C01814=1073.007,225.307,-82.417,174.106,27.682,154.920
C01815=1073.013,225.555,-82.444,174.109,27.687,154.920
C01816=1073.019,225.804,-82.469,174.111,27.690,154.921
C01817=1073.025,226.052,-82.496,174.113,27.694,154.921
C01818=1073.031,226.301,-82.522,174.116,27.698,154.922
C01819=1073.036,226.549,-82.549,174.118,27.702,154.923
C01820=1073.043,226.798,-82.574,174.120,27.706,154.923
C01821=1073.048,227.046,-82.601,174.123,27.710,154.924
C01822=1073.054,227.295,-82.627,174.125,27.713,154.924
C01823=1073.060,227.544,-82.652,174.127,27.717,154.925
C01824=1073.066,227.792,-82.679,174.129,27.721,154.926
C01825=1073.072,228.041,-82.705,174.131,27.725,154.926
C01826=1073.078,228.289,-82.731,174.133,27.729,154.927
C01827=1073.084,228.538,-82.757,174.136,27.733,154.927
C01828=1073.089,228.787,-82.783,174.138,27.736,154.928
C01829=1073.096,229.036,-82.810,174.140,27.740,154.929
C01830=1073.102,229.285,-82.835,174.143,27.744,154.929
C01831=1073.107,229.533,-82.862,174.145,27.748,154.930
C01832=1073.113,229.782,-82.888,174.147,27.752,154.930
C01833=1073.119,230.030,-82.914,174.150,27.755,154.931
C01834=1073.125,230.278,-82.941,174.152,27.760,154.932
C01835=1073.131,230.527,-82.967,174.154,27.764,154.932
C01836=1073.136,230.776,-82.993,174.156,27.768,154.933
C01837=1073.142,231.024,-83.020,174.158,27.771,154.933
C01838=1073.148,231.273,-83.046,174.160,27.775,154.934
C01839=1073.153,231.521,-83.073,174.163,27.779,154.935
C01840=1073.159,231.770,-83.099,174.165,27.782,154.935
C01841=1073.165,232.018,-83.126,174.167,27.787,154.936
C01842=1073.170,232.267,-83.152,174.169,27.791,154.936
C01843=1073.177,232.515,-83.178,174.172,27.795,154.937
C01844=1073.183,232.764,-83.205,174.174,27.798,154.938
C01845=1073.189,233.013,-83.231,174.176,27.802,154.938
C01846=1073.195,233.262,-83.257,174.179,27.806,154.939
C01847=1073.200,233.510,-83.284,174.181,27.810,154.939
C01848=1073.206,233.758,-83.311,174.183,27.814,154.940
C01849=1073.212,234.007,-83.337,174.186,27.818,154.941
C01850=1073.218,234.255,-83.364,174.188,27.821,154.941
C01851=1073.223,234.504,-83.390,174.190,27.825,154.942
C01852=1073.229,234.752,-83.417,174.193,27.829,154.943
C01853=1073.235,235.001,-83.443,174.195,27.833,154.943
C01854=1073.244,235.416,-83.489,174.198,27.839,154.944
C01855=1073.254,235.831,-83.533,174.202,27.846,154.945
C01856=1073.264,236.245,-83.577,174.206,27.852,154.946
C01857=1073.273,236.660,-83.623,174.210,27.859,154.947
C01858=1073.279,236.908,-83.649,174.212,27.863,154.948
C01859=1073.285,237.157,-83.676,174.214,27.867,154.948
C01860=1073.291,237.405,-83.703,174.217,27.871,154.949
C01861=1073.296,237.653,-83.729,174.219,27.874,154.950
C01862=1073.303,237.902,-83.756,174.221,27.878,154.950
C01863=1073.309,238.151,-83.783,174.224,27.882,154.951
C01864=1073.314,238.399,-83.809,174.226,27.886,154.951
C01865=1073.320,238.648,-83.836,174.228,27.890,154.952
C01866=1073.327,238.897,-83.863,174.231,27.894,154.953
C01867=1073.332,239.145,-83.890,174.233,27.897,154.953
C01868=1073.337,239.394,-83.917,174.235,27.901,154.954
C01869=1073.343,239.642,-83.944,174.238,27.905,154.954
C01870=1073.350,239.891,-83.971,174.240,27.909,154.955
C01871=1073.355,240.139,-83.997,174.242,27.913,154.956
C01872=1073.361,240.387,-84.025,174.245,27.917,154.956
C01873=1073.367,240.636,-84.051,174.247,27.920,154.957
C01874=1073.373,240.885,-84.079,174.249,27.924,154.957
C01875=1073.379,241.133,-84.106,174.252,27.928,154.958
C01876=1073.384,241.382,-84.132,174.254,27.932,154.959
C01877=1073.390,241.629,-84.160,174.257,27.936,154.959
C01878=1073.397,241.878,-84.187,174.259,27.940,154.960
C01879=1073.402,242.127,-84.214,174.261,27.943,154.960
C01880=1073.408,242.375,-84.241,174.264,27.947,154.961
C01881=1073.414,242.624,-84.268,174.266,27.951,154.962
C01882=1073.420,242.872,-84.295,174.268,27.955,154.962
C01883=1073.425,243.121,-84.322,174.271,27.959,154.963
C01884=1073.431,243.369,-84.350,174.273,27.963,154.963
C01885=1073.438,243.618,-84.377,174.275,27.967,154.964
C01886=1073.443,243.866,-84.404,174.278,27.971,154.965
C01887=1073.449,244.114,-84.431,174.280,27.975,154.965
C01888=1073.454,244.364,-84.459,174.282,27.978,154.966
C01889=1073.460,244.612,-84.485,174.285,27.982,154.966
C01890=1073.466,244.860,-84.513,174.287,27.986,154.967
C01891=1073.472,245.109,-84.540,174.289,27.990,154.968
C01892=1073.478,245.357,-84.568,174.292,27.994,154.968
C01893=1073.483,245.605,-84.595,174.294,27.998,154.969
C01894=1073.490,245.854,-84.623,174.296,28.002,154.970
C01895=1073.495,246.103,-84.650,174.300,28.005,154.970
C01896=1073.500,246.351,-84.677,174.302,28.009,154.971
C01897=1073.507,246.599,-84.704,174.304,28.013,154.971
C01898=1073.512,246.848,-84.732,174.307,28.017,154.972
C01899=1073.518,247.096,-84.759,174.309,28.021,154.972
C01900=1073.524,247.344,-84.787,174.312,28.025,154.973
C01901=1073.529,247.593,-84.815,174.314,28.029,154.974
C01902=1073.535,247.841,-84.842,174.316,28.033,154.974
C01903=1073.541,248.090,-84.869,174.319,28.036,154.975
C01904=1073.547,248.338,-84.897,174.321,28.040,154.976
C01905=1073.552,248.587,-84.924,174.323,28.045,154.976
C01906=1073.562,248.995,-84.970,174.327,28.051,154.977
C01907=1073.571,249.403,-85.015,174.331,28.057,154.978
C01908=1073.581,249.812,-85.061,174.335,28.064,154.979
C01909=1073.590,250.219,-85.107,174.339,28.070,154.980
C01910=1073.595,250.468,-85.134,174.341,28.074,154.981
C01911=1073.601,250.716,-85.161,174.344,28.078,154.982
C01912=1073.607,250.965,-85.190,174.346,28.082,154.982
C01913=1073.613,251.213,-85.218,174.348,28.086,154.983
C01914=1073.619,251.462,-85.245,174.351,28.090,154.983
C01915=1073.624,251.710,-85.273,174.353,28.094,154.984
C01916=1073.630,251.958,-85.301,174.356,28.097,154.985
C01917=1073.636,252.206,-85.328,174.359,28.101,154.985
C01918=1073.641,252.455,-85.356,174.361,28.105,154.986
C01919=1073.647,252.704,-85.384,174.363,28.109,154.986
C01920=1073.653,252.951,-85.411,174.366,28.113,154.987
C01921=1073.659,253.200,-85.440,174.368,28.117,154.988
C01922=1073.665,253.448,-85.468,174.371,28.121,154.988
C01923=1073.671,253.697,-85.495,174.373,28.125,154.989
C01924=1073.677,253.945,-85.523,174.375,28.128,154.989
C01925=1073.683,254.193,-85.552,174.378,28.132,154.990
C01926=1073.688,254.442,-85.579,174.380,28.136,154.991
C01927=1073.694,254.691,-85.607,174.383,28.140,154.991
C01928=1073.700,254.939,-85.635,174.386,28.144,154.992
C01929=1073.706,255.187,-85.663,174.388,28.148,154.993
C01930=1073.712,255.436,-85.691,174.390,28.152,154.993
C01931=1073.718,255.684,-85.719,174.393,28.156,154.994
C01932=1073.724,255.933,-85.747,174.395,28.160,154.994
C01933=1073.729,256.181,-85.775,174.398,28.164,154.995
C01934=1073.735,256.429,-85.803,174.400,28.167,154.996
C01935=1073.741,256.677,-85.831,174.402,28.171,154.996
C01936=1073.747,256.926,-85.859,174.406,28.175,154.997
C01937=1073.753,257.175,-85.887,174.408,28.179,154.997
C01938=1073.758,257.423,-85.915,174.410,28.183,154.998
C01939=1073.765,257.671,-85.944,174.413,28.187,154.999
C01940=1073.771,257.919,-85.972,174.415,28.190,154.999
C01941=1073.776,258.167,-86.000,174.418,28.194,155.000
C01942=1073.782,258.416,-86.028,174.420,28.198,155.000
C01943=1073.788,258.664,-86.056,174.422,28.202,155.001
C01944=1073.794,258.913,-86.084,174.426,28.206,155.002
C01945=1073.800,259.161,-86.112,174.428,28.210,155.002
C01946=1073.806,259.409,-86.141,174.430,28.214,155.003
C01947=1073.812,259.657,-86.169,174.433,28.217,155.003
C01948=1073.818,259.906,-86.198,174.435,28.221,155.004
C01949=1073.824,260.154,-86.225,174.438,28.225,155.005
C01950=1073.830,260.403,-86.253,174.440,28.229,155.005
C01951=1073.836,260.651,-86.282,174.443,28.233,155.006
C01952=1073.842,260.899,-86.310,174.446,28.237,155.006
C01953=1073.847,261.148,-86.339,174.448,28.241,155.007
C01954=1073.854,261.396,-86.368,174.450,28.245,155.008
C01955=1073.860,261.644,-86.395,174.453,28.248,155.008
C01956=1073.866,261.892,-86.423,174.455,28.252,155.009
C01957=1073.872,262.140,-86.452,174.459,28.256,155.009
C01958=1073.881,262.547,-86.499,174.463,28.262,155.010
C01959=1073.891,262.952,-86.545,174.467,28.268,155.011
C01960=1073.902,263.357,-86.591,174.471,28.275,155.012
C01961=1073.911,263.764,-86.638,174.475,28.281,155.013
C01962=1073.917,264.011,-86.666,174.477,28.285,155.014
C01963=1073.923,264.260,-86.695,174.480,28.289,155.015
C01964=1073.929,264.508,-86.724,174.483,28.293,155.015
C01965=1073.934,264.756,-86.752,174.485,28.297,155.016
C01966=1073.941,265.004,-86.781,174.488,28.300,155.016
C01967=1073.946,265.253,-86.810,174.490,28.304,155.017
C01968=1073.952,265.502,-86.839,174.493,28.309,155.018
C01969=1073.957,265.750,-86.867,174.496,28.312,155.018
C01970=1073.964,265.998,-86.896,174.498,28.316,155.019
C01971=1073.970,266.246,-86.925,174.500,28.320,155.019
C01972=1073.976,266.495,-86.953,174.503,28.324,155.020
C01973=1073.981,266.742,-86.982,174.505,28.328,155.021
C01974=1073.987,266.991,-87.011,174.508,28.332,155.021
C01975=1073.993,267.239,-87.040,174.511,28.336,155.022
C01976=1073.999,267.487,-87.069,174.513,28.340,155.023
C01977=1074.005,267.736,-87.097,174.516,28.343,155.023
C01978=1074.010,267.984,-87.126,174.518,28.347,155.024
C01979=1074.016,268.232,-87.155,174.521,28.352,155.025
C01980=1074.022,268.481,-87.184,174.524,28.355,155.025
C01981=1074.028,268.729,-87.213,174.526,28.359,155.026
C01982=1074.035,268.977,-87.242,174.529,28.363,155.026
C01983=1074.040,269.226,-87.272,174.532,28.367,155.027
C01984=1074.046,269.474,-87.299,174.534,28.371,155.028
C01985=1074.052,269.722,-87.329,174.537,28.375,155.028
C01986=1074.057,269.970,-87.358,174.539,28.379,155.029
C01987=1074.064,270.218,-87.387,174.542,28.383,155.029
C01988=1074.070,270.466,-87.416,174.545,28.387,155.030
C01989=1074.076,270.715,-87.445,174.547,28.391,155.031
C01990=1074.081,270.963,-87.474,174.550,28.395,155.031
C01991=1074.087,271.211,-87.503,174.552,28.399,155.032
C01992=1074.092,271.459,-87.533,174.555,28.402,155.033
C01993=1074.099,271.708,-87.562,174.558,28.406,155.033
C01994=1074.105,271.956,-87.591,174.560,28.410,155.034
C01995=1074.110,272.204,-87.620,174.563,28.414,155.034
C01996=1074.117,272.452,-87.649,174.565,28.418,155.035
C01997=1074.123,272.700,-87.678,174.568,28.423,155.036
C01998=1074.128,272.949,-87.708,174.571,28.426,155.036
C01999=1074.134,273.196,-87.737,174.573,28.430,155.037
C02000=1074.140,273.445,-87.766,174.576,28.434,155.038
C02001=1074.146,273.693,-87.795,174.579,28.438,155.038
C02002=1074.151,273.941,-87.825,174.581,28.442,155.039
C02003=1074.158,274.189,-87.854,174.584,28.446,155.040
C02004=1074.163,274.438,-87.884,174.586,28.450,155.040
C02005=1074.169,274.686,-87.913,174.589,28.454,155.041
C02006=1074.175,274.934,-87.942,174.592,28.458,155.041
C02007=1074.181,275.183,-87.971,174.594,28.462,155.042
C02008=1074.187,275.431,-88.001,174.597,28.466,155.043
C02009=1074.193,275.679,-88.030,174.600,28.470,155.043
C02010=1074.202,276.088,-88.078,174.604,28.476,155.044
C02011=1074.212,276.496,-88.128,174.609,28.483,155.045
C02012=1074.222,276.906,-88.176,174.613,28.489,155.046
C02013=1074.232,277.314,-88.224,174.617,28.496,155.047
C02014=1074.237,277.562,-88.254,174.620,28.500,155.048
C02015=1074.243,277.811,-88.283,174.623,28.504,155.049
C02016=1074.249,278.058,-88.313,174.625,28.508,155.049
C02017=1074.255,278.307,-88.343,174.627,28.512,155.050
C02018=1074.261,278.555,-88.372,174.631,28.516,155.051
C02019=1074.267,278.803,-88.402,174.633,28.520,155.051
C02020=1074.272,279.051,-88.432,174.636,28.524,155.052
C02021=1074.279,279.299,-88.461,174.639,28.528,155.052
C02022=1074.284,279.547,-88.491,174.641,28.532,155.053
C02023=1074.290,279.796,-88.521,174.644,28.536,155.054
C02024=1074.296,280.044,-88.550,174.646,28.540,155.054
C02025=1074.303,280.292,-88.581,174.650,28.544,155.055
C02026=1074.308,280.541,-88.610,174.652,28.548,155.056
C02027=1074.315,280.788,-88.640,174.654,28.552,155.056
C02028=1074.320,281.037,-88.670,174.658,28.556,155.057
C02029=1074.326,281.285,-88.699,174.660,28.560,155.058
C02030=1074.332,281.533,-88.730,174.663,28.564,155.058
C02031=1074.337,281.781,-88.759,174.666,28.568,155.059
C02032=1074.344,282.029,-88.789,174.668,28.572,155.060
C02033=1074.349,282.277,-88.819,174.671,28.576,155.060
C02034=1074.355,282.525,-88.849,174.674,28.580,155.061
C02035=1074.361,282.773,-88.879,174.676,28.584,155.062
C02036=1074.366,283.021,-88.909,174.679,28.588,155.062
C02037=1074.372,283.269,-88.939,174.681,28.592,155.063
C02038=1074.378,283.517,-88.968,174.685,28.596,155.063
C02039=1074.385,283.766,-88.999,174.687,28.600,155.064
C02040=1074.391,284.014,-89.029,174.689,28.605,155.065
C02041=1074.396,284.262,-89.059,174.693,28.609,155.066
C02042=1074.402,284.510,-89.089,174.695,28.613,155.066
C02043=1074.407,284.758,-89.119,174.698,28.617,155.067
C02044=1074.413,285.006,-89.149,174.701,28.621,155.067
C02045=1074.419,285.254,-89.180,174.703,28.625,155.068
C02046=1074.426,285.502,-89.210,174.707,28.629,155.069
C02047=1074.432,285.751,-89.240,174.709,28.633,155.069
C02048=1074.438,285.999,-89.270,174.712,28.637,155.070
C02049=1074.443,286.246,-89.300,174.715,28.641,155.071
C02050=1074.449,286.494,-89.331,174.717,28.645,155.071
C02051=1074.455,286.743,-89.361,174.720,28.649,155.072
C02052=1074.461,286.991,-89.391,174.723,28.653,155.073
C02053=1074.467,287.239,-89.421,174.726,28.657,155.073
C02054=1074.473,287.487,-89.452,174.728,28.661,155.074
C02055=1074.479,287.735,-89.482,174.731,28.665,155.075
C02056=1074.485,287.984,-89.512,174.734,28.669,155.075
C02057=1074.491,288.231,-89.542,174.736,28.673,155.076
C02058=1074.497,288.479,-89.572,174.740,28.677,155.077
C02059=1074.503,288.727,-89.602,174.742,28.681,155.077
C02060=1074.509,288.975,-89.633,174.745,28.685,155.078
C02061=1074.515,289.223,-89.664,174.748,28.689,155.078
C02062=1074.525,289.642,-89.715,174.753,28.696,155.080
C02063=1074.535,290.061,-89.766,174.757,28.703,155.081
C02064=1074.545,290.480,-89.818,174.762,28.710,155.082
C02065=1074.555,290.899,-89.869,174.767,28.717,155.083
C02066=1074.560,291.147,-89.900,174.769,28.721,155.084
C02067=1074.566,291.396,-89.931,174.772,28.725,155.084
C02068=1074.572,291.643,-89.961,174.775,28.729,155.085
C02069=1074.578,291.891,-89.992,174.777,28.734,155.086
C02070=1074.585,292.139,-90.023,174.781,28.738,155.086
C02071=1074.591,292.387,-90.053,174.783,28.742,155.087
C02072=1074.596,292.635,-90.084,174.786,28.746,155.088
C02073=1074.602,292.883,-90.115,174.789,28.750,155.088
C02074=1074.608,293.131,-90.145,174.791,28.754,155.089
C02075=1074.614,293.379,-90.176,174.795,28.758,155.090
C02076=1074.620,293.626,-90.207,174.797,28.762,155.090
C02077=1074.626,293.875,-90.238,174.800,28.766,155.091
C02078=1074.631,294.123,-90.268,174.803,28.770,155.092
C02079=1074.638,294.372,-90.299,174.806,28.775,155.092
C02080=1074.644,294.619,-90.330,174.809,28.779,155.093
C02081=1074.650,294.867,-90.361,174.811,28.783,155.094
C02082=1074.655,295.115,-90.392,174.814,28.787,155.094
C02083=1074.662,295.363,-90.423,174.817,28.792,155.095
C02084=1074.667,295.610,-90.453,174.820,28.796,155.096
C02085=1074.673,295.859,-90.485,174.823,28.800,155.096
C02086=1074.679,296.107,-90.516,174.826,28.804,155.097
C02087=1074.686,296.355,-90.546,174.828,28.808,155.098
C02088=1074.691,296.603,-90.577,174.831,28.812,155.099
C02089=1074.697,296.850,-90.608,174.834,28.816,155.099
C02090=1074.703,297.099,-90.639,174.837,28.820,155.100
C02091=1074.709,297.346,-90.671,174.840,28.825,155.101
C02092=1074.715,297.595,-90.702,174.842,28.829,155.101
C02093=1074.720,297.842,-90.733,174.846,28.833,155.102
C02094=1074.727,298.091,-90.764,174.848,28.837,155.103
C02095=1074.732,298.339,-90.796,174.852,28.842,155.103
C02096=1074.738,298.586,-90.826,174.854,28.846,155.104
C02097=1074.744,298.835,-90.858,174.857,28.850,155.105
C02098=1074.750,299.082,-90.888,174.860,28.855,155.106
C02099=1074.755,299.330,-90.920,174.862,28.858,155.106
C02100=1074.761,299.579,-90.951,174.866,28.863,155.107
C02101=1074.767,299.826,-90.982,174.868,28.867,155.108
C02102=1074.773,300.074,-91.014,174.871,28.872,155.108
C02103=1074.779,300.322,-91.045,174.874,28.876,155.109
C02104=1074.785,300.570,-91.077,174.877,28.880,155.110
C02105=1074.790,300.818,-91.108,174.880,28.884,155.110
C02106=1074.796,301.065,-91.139,174.883,28.889,155.111
C02107=1074.802,301.314,-91.171,174.885,28.893,155.112
C02108=1074.807,301.561,-91.202,174.889,28.897,155.113
C02109=1074.814,301.810,-91.233,174.891,28.901,155.113
C02110=1074.819,302.057,-91.265,174.894,28.906,155.114
C02111=1074.825,302.305,-91.297,174.897,28.910,155.115
C02112=1074.831,302.553,-91.328,174.900,28.915,155.115
C02113=1074.837,302.801,-91.360,174.903,28.918,155.116
C02114=1074.842,303.017,-91.387,174.905,28.922,155.117
C02115=1074.847,303.235,-91.415,174.908,28.926,155.117
C02116=1074.852,303.451,-91.442,174.910,28.930,155.118
C02117=1074.858,303.668,-91.470,174.913,28.934,155.119
C02118=1074.863,303.885,-91.497,174.916,28.938,155.119
C02119=1074.868,304.102,-91.525,174.919,28.941,155.120
C02120=1074.873,304.318,-91.553,174.921,28.945,155.120
C02121=1074.879,304.535,-91.580,174.923,28.949,155.121
C02122=1074.884,304.783,-91.612,174.926,28.953,155.122
C02123=1074.890,305.031,-91.644,174.929,28.957,155.123
C02124=1074.897,305.279,-91.675,174.932,28.961,155.123
C02125=1074.902,305.526,-91.707,174.935,28.966,155.124
C02126=1074.908,305.775,-91.739,174.938,28.970,155.125
C02127=1074.914,306.022,-91.770,174.941,28.975,155.125
C02128=1074.920,306.270,-91.802,174.943,28.979,155.126
C02129=1074.926,306.518,-91.834,174.947,28.983,155.127
C02130=1074.932,306.766,-91.866,174.950,28.988,155.128
C02131=1074.938,307.014,-91.897,174.952,28.992,155.128
C02132=1074.944,307.262,-91.929,174.956,28.996,155.129
C02133=1074.950,307.509,-91.961,174.958,29.000,155.130
C02134=1074.956,307.758,-91.993,174.962,29.005,155.130
C02135=1074.962,308.005,-92.024,174.964,29.009,155.131
C02136=1074.968,308.252,-92.057,174.967,29.013,155.132
C02137=1074.974,308.501,-92.089,174.970,29.018,155.133
C02138=1074.980,308.749,-92.121,174.973,29.022,155.133
C02139=1074.986,308.996,-92.152,174.977,29.027,155.134
C02140=1074.992,309.244,-92.184,174.979,29.030,155.135
C02141=1074.998,309.492,-92.216,174.982,29.035,155.136
C02142=1075.004,309.740,-92.249,174.985,29.039,155.136
C02143=1075.011,309.987,-92.280,174.988,29.044,155.137
C02144=1075.017,310.235,-92.312,174.991,29.048,155.138
C02145=1075.023,310.484,-92.344,174.994,29.052,155.138
C02146=1075.029,310.731,-92.377,174.998,29.057,155.139
C02147=1075.035,310.979,-92.409,175.000,29.061,155.140
C02148=1075.040,311.227,-92.440,175.003,29.065,155.141
C02149=1075.047,311.474,-92.472,175.006,29.070,155.141
C02150=1075.053,311.722,-92.504,175.009,29.074,155.142
C02151=1075.059,311.971,-92.536,175.013,29.078,155.143
C02152=1075.066,312.218,-92.569,175.015,29.083,155.144
C02153=1075.072,312.466,-92.601,175.018,29.087,155.144
C02154=1075.077,312.714,-92.633,175.021,29.091,155.145
C02155=1075.084,312.961,-92.665,175.024,29.096,155.146
C02156=1075.090,313.209,-92.697,175.028,29.100,155.146
C02157=1075.096,313.457,-92.730,175.030,29.104,155.147
C02158=1075.102,313.705,-92.762,175.033,29.109,155.148
C02159=1075.109,313.953,-92.795,175.036,29.113,155.149
C02160=1075.115,314.201,-92.827,175.039,29.118,155.149
C02161=1075.121,314.449,-92.859,175.043,29.122,155.150
C02162=1075.127,314.697,-92.891,175.045,29.127,155.151
C02163=1075.132,314.944,-92.924,175.048,29.131,155.152
C02164=1075.138,315.192,-92.956,175.051,29.136,155.152
C02165=1075.144,315.440,-92.989,175.054,29.140,155.153
C02166=1075.150,315.687,-93.022,175.058,29.145,155.154
C02167=1075.156,315.936,-93.054,175.060,29.149,155.155
C02168=1075.161,316.183,-93.087,175.063,29.154,155.156
C02169=1075.168,316.431,-93.120,175.066,29.158,155.156
C02170=1075.174,316.681,-93.152,175.069,29.163,155.157
C02171=1075.180,316.930,-93.185,175.073,29.168,155.158
C02172=1075.185,317.180,-93.218,175.075,29.172,155.159
C02173=1075.191,317.429,-93.250,175.078,29.177,155.159
C02174=1075.197,317.677,-93.283,175.082,29.181,155.160
C02175=1075.203,317.925,-93.317,175.084,29.186,155.161
C02176=1075.209,318.173,-93.349,175.088,29.190,155.162
C02177=1075.215,318.420,-93.382,175.091,29.195,155.163
C02178=1075.221,318.669,-93.415,175.093,29.199,155.163
C02179=1075.227,318.916,-93.447,175.097,29.204,155.164
C02180=1075.233,319.164,-93.480,175.100,29.209,155.165
C02181=1075.239,319.412,-93.513,175.103,29.213,155.166
C02182=1075.245,319.659,-93.546,175.106,29.218,155.167
C02183=1075.251,319.907,-93.580,175.108,29.222,155.167
C02184=1075.257,320.155,-93.612,175.112,29.227,155.168
C02185=1075.263,320.403,-93.644,175.115,29.232,155.169
C02186=1075.268,320.651,-93.678,175.118,29.236,155.170
C02187=1075.275,320.899,-93.710,175.121,29.241,155.170
C02188=1075.280,321.146,-93.744,175.124,29.246,155.171
C02189=1075.287,321.394,-93.776,175.127,29.250,155.172
C02190=1075.292,321.611,-93.805,175.130,29.254,155.173
C02191=1075.297,321.829,-93.835,175.133,29.258,155.173
C02192=1075.302,322.046,-93.863,175.135,29.262,155.174
C02193=1075.308,322.263,-93.893,175.138,29.266,155.175
C02194=1075.313,322.480,-93.921,175.141,29.270,155.175
C02195=1075.318,322.698,-93.951,175.144,29.274,155.176
C02196=1075.324,322.916,-93.980,175.146,29.279,155.177
C02197=1075.329,323.133,-94.009,175.149,29.282,155.178
C02198=1075.335,323.380,-94.041,175.152,29.287,155.178
C02199=1075.341,323.628,-94.075,175.155,29.292,155.179
C02200=1075.347,323.876,-94.107,175.158,29.297,155.180
C02201=1075.353,324.125,-94.141,175.161,29.301,155.181
C02202=1075.360,324.372,-94.175,175.165,29.306,155.182
C02203=1075.365,324.619,-94.208,175.168,29.310,155.182
C02204=1075.371,324.867,-94.241,175.170,29.315,155.183
C02205=1075.377,325.115,-94.274,175.174,29.320,155.184
C02206=1075.383,325.363,-94.307,175.177,29.324,155.185
C02207=1075.390,325.611,-94.341,175.180,29.329,155.186
C02208=1075.396,325.858,-94.374,175.183,29.334,155.187
C02209=1075.402,326.106,-94.407,175.186,29.339,155.187
C02210=1075.408,326.353,-94.441,175.190,29.343,155.188
C02211=1075.414,326.601,-94.474,175.192,29.347,155.189
C02212=1075.421,326.849,-94.507,175.196,29.353,155.190
C02213=1075.426,327.096,-94.541,175.199,29.357,155.191
C02214=1075.433,327.344,-94.574,175.202,29.362,155.191
C02215=1075.438,327.592,-94.607,175.205,29.367,155.192
C02216=1075.446,327.840,-94.641,175.208,29.371,155.193
C02217=1075.451,328.088,-94.675,175.212,29.376,155.194
C02218=1075.458,328.335,-94.708,175.215,29.381,155.195
C02219=1075.463,328.582,-94.741,175.217,29.385,155.195
C02220=1075.470,328.830,-94.776,175.221,29.390,155.196
C02221=1075.476,329.078,-94.808,175.224,29.395,155.197
C02222=1075.482,329.325,-94.843,175.228,29.400,155.198
C02223=1075.489,329.574,-94.876,175.231,29.404,155.199
C02224=1075.495,329.821,-94.910,175.233,29.409,155.200
C02225=1075.501,330.068,-94.942,175.237,29.414,155.200
C02226=1075.506,330.283,-94.972,175.239,29.418,155.201
C02227=1075.512,330.500,-95.001,175.243,29.422,155.202
C02228=1075.518,330.714,-95.031,175.245,29.426,155.203
C02229=1075.522,330.930,-95.060,175.248,29.430,155.203
C02230=1075.528,331.145,-95.089,175.251,29.434,155.204
C02231=1075.534,331.359,-95.118,175.254,29.439,155.205
C02232=1075.538,331.575,-95.148,175.256,29.443,155.206
C02233=1075.543,331.790,-95.178,175.259,29.447,155.206
C02234=1075.551,332.038,-95.211,175.262,29.452,155.207
C02235=1075.556,332.286,-95.245,175.265,29.457,155.208
C02236=1075.562,332.533,-95.279,175.269,29.462,155.209
C02237=1075.568,332.781,-95.313,175.272,29.467,155.210
C02238=1075.574,333.028,-95.347,175.275,29.472,155.211
C02239=1075.580,333.276,-95.381,175.278,29.476,155.211
C02240=1075.586,333.524,-95.415,175.281,29.481,155.212
C02241=1075.592,333.771,-95.449,175.285,29.486,155.213
C02242=1075.598,334.019,-95.483,175.288,29.491,155.214
C02243=1075.605,334.267,-95.518,175.292,29.496,155.215
C02244=1075.610,334.514,-95.552,175.294,29.501,155.216
C02245=1075.616,334.761,-95.586,175.297,29.506,155.217
C02246=1075.622,335.010,-95.619,175.301,29.511,155.218
C02247=1075.628,335.257,-95.653,175.304,29.516,155.218
C02248=1075.635,335.505,-95.687,175.308,29.521,155.219
C02249=1075.641,335.752,-95.721,175.311,29.526,155.220
C02250=1075.648,336.000,-95.756,175.313,29.531,155.221
C02251=1075.654,336.247,-95.790,175.317,29.536,155.222
C02252=1075.660,336.495,-95.824,175.320,29.541,155.223
C02253=1075.666,336.743,-95.858,175.324,29.546,155.224
C02254=1075.672,336.991,-95.893,175.327,29.550,155.224
C02255=1075.679,337.237,-95.927,175.330,29.556,155.225
C02256=1075.685,337.485,-95.962,175.334,29.561,155.226
C02257=1075.691,337.732,-95.996,175.336,29.565,155.227
C02258=1075.697,337.980,-96.030,175.340,29.571,155.228
C02259=1075.703,338.228,-96.065,175.343,29.576,155.229
C02260=1075.708,338.475,-96.099,175.346,29.581,155.230
C02261=1075.715,338.723,-96.133,175.350,29.586,155.231
C02262=1075.721,338.970,-96.168,175.353,29.591,155.232
C02263=1075.727,339.218,-96.203,175.357,29.596,155.233
C02264=1075.733,339.466,-96.237,175.360,29.601,155.233
C02265=1075.739,339.714,-96.272,175.362,29.606,155.234
C02266=1075.745,339.960,-96.306,175.366,29.611,155.235
C02267=1075.752,340.208,-96.341,175.369,29.616,155.236
C02268=1075.758,340.456,-96.375,175.373,29.622,155.237
C02269=1075.764,340.703,-96.411,175.376,29.627,155.238
C02270=1075.770,340.951,-96.445,175.379,29.632,155.239
C02271=1075.776,341.198,-96.479,175.383,29.637,155.240
C02272=1075.783,341.446,-96.514,175.386,29.642,155.241
C02273=1075.788,341.693,-96.549,175.390,29.647,155.242
C02274=1075.795,341.941,-96.584,175.393,29.652,155.243
C02275=1075.801,342.189,-96.618,175.396,29.658,155.244
C02276=1075.807,342.436,-96.652,175.399,29.662,155.245
C02277=1075.813,342.684,-96.688,175.402,29.668,155.246
C02278=1075.819,342.932,-96.723,175.406,29.673,155.247
C02279=1075.826,343.178,-96.757,175.409,29.678,155.247
C02280=1075.832,343.426,-96.792,175.412,29.683,155.248
C02281=1075.838,343.674,-96.828,175.416,29.689,155.249
C02282=1075.843,343.886,-96.858,175.419,29.693,155.250
C02283=1075.849,344.099,-96.887,175.422,29.698,155.251
C02284=1075.854,344.311,-96.917,175.424,29.702,155.252
C02285=1075.859,344.524,-96.947,175.428,29.706,155.253
C02286=1075.865,344.736,-96.978,175.430,29.711,155.253
C02287=1075.869,344.949,-97.007,175.434,29.716,155.254
C02288=1075.875,345.162,-97.037,175.436,29.720,155.255
C02289=1075.880,345.374,-97.067,175.439,29.724,155.256
C02290=1075.886,345.621,-97.103,175.442,29.730,155.257
C02291=1075.893,345.869,-97.137,175.445,29.735,155.258
C02292=1075.899,346.116,-97.172,175.449,29.741,155.259
C02293=1075.905,346.364,-97.208,175.452,29.746,155.260
C02294=1075.912,346.611,-97.243,175.456,29.751,155.261
C02295=1075.917,346.858,-97.278,175.459,29.757,155.262
C02296=1075.923,347.106,-97.313,175.462,29.762,155.263
C02297=1075.930,347.354,-97.349,175.466,29.767,155.264
C02298=1075.936,347.601,-97.384,175.469,29.772,155.265
C02299=1075.942,347.848,-97.419,175.473,29.778,155.266
C02300=1075.948,348.096,-97.455,175.476,29.783,155.267
C02301=1075.955,348.343,-97.490,175.479,29.789,155.268
C02302=1075.961,348.591,-97.526,175.483,29.794,155.269
C02303=1075.968,348.838,-97.561,175.486,29.800,155.270
C02304=1075.973,349.085,-97.596,175.490,29.805,155.270
C02305=1075.979,349.333,-97.632,175.493,29.810,155.272
C02306=1075.986,349.580,-97.667,175.496,29.816,155.273
C02307=1075.992,349.828,-97.703,175.500,29.821,155.274
C02308=1075.999,350.075,-97.738,175.503,29.826,155.274
C02309=1076.004,350.322,-97.773,175.507,29.832,155.276
C02310=1076.010,350.570,-97.809,175.510,29.837,155.277
C02311=1076.017,350.817,-97.844,175.513,29.843,155.278
C02312=1076.023,351.065,-97.880,175.517,29.849,155.279
C02313=1076.030,351.312,-97.915,175.520,29.854,155.280
C02314=1076.036,351.560,-97.951,175.524,29.859,155.281
C02315=1076.042,351.807,-97.987,175.528,29.865,155.282
C02316=1076.048,352.054,-98.022,175.531,29.870,155.283
C02317=1076.054,352.301,-98.058,175.535,29.876,155.284
C02318=1076.060,352.549,-98.093,175.538,29.881,155.285
C02319=1076.066,352.797,-98.129,175.542,29.887,155.286
C02320=1076.073,353.043,-98.165,175.545,29.893,155.287
C02321=1076.079,353.291,-98.201,175.548,29.898,155.288
C02322=1076.085,353.539,-98.236,175.552,29.904,155.289
C02323=1076.092,353.786,-98.273,175.555,29.909,155.290
C02324=1076.098,354.033,-98.309,175.559,29.915,155.291
C02325=1076.104,354.281,-98.344,175.562,29.921,155.292
C02326=1076.110,354.527,-98.380,175.565,29.926,155.293
C02327=1076.116,354.775,-98.416,175.569,29.932,155.294
C02328=1076.123,355.022,-98.452,175.572,29.937,155.295
C02329=1076.129,355.270,-98.488,175.576,29.943,155.296
C02330=1076.135,355.517,-98.524,175.580,29.949,155.297
C02331=1076.141,355.764,-98.560,175.583,29.955,155.298
C02332=1076.147,356.011,-98.596,175.587,29.960,155.299
C02333=1076.153,356.259,-98.632,175.590,29.966,155.300
C02334=1076.160,356.506,-98.668,175.593,29.972,155.302
C02335=1076.166,356.753,-98.704,175.597,29.977,155.303
C02336=1076.173,357.001,-98.740,175.600,29.983,155.304
C02337=1076.179,357.248,-98.777,175.604,29.989,155.305
C02338=1076.185,357.463,-98.808,175.607,29.994,155.306
C02339=1076.190,357.677,-98.839,175.611,29.999,155.307
C02340=1076.195,357.891,-98.871,175.613,30.004,155.307
C02341=1076.201,358.105,-98.901,175.617,30.009,155.308
C02342=1076.207,358.319,-98.933,175.619,30.013,155.309
C02343=1076.212,358.534,-98.965,175.623,30.018,155.310
C02344=1076.217,358.747,-98.996,175.626,30.024,155.311
C02345=1076.223,358.962,-99.027,175.628,30.029,155.312
C02346=1076.230,359.209,-99.064,175.632,30.034,155.313
C02347=1076.236,359.457,-99.100,175.635,30.040,155.314
C02348=1076.242,359.704,-99.137,175.640,30.046,155.315
C02349=1076.248,359.951,-99.172,175.643,30.052,155.317
C02350=1076.255,360.198,-99.209,175.646,30.058,155.318
C02351=1076.260,360.446,-99.246,175.650,30.063,155.319
C02352=1076.267,360.693,-99.282,175.653,30.070,155.320
C02353=1076.273,360.940,-99.319,175.657,30.076,155.321
C02354=1076.279,361.187,-99.355,175.661,30.081,155.322
C02355=1076.286,361.434,-99.392,175.664,30.087,155.323
C02356=1076.293,361.682,-99.429,175.668,30.093,155.324
C02357=1076.299,361.929,-99.465,175.671,30.099,155.326
C02358=1076.305,362.176,-99.501,175.675,30.105,155.327
C02359=1076.311,362.423,-99.538,175.679,30.111,155.328
C02360=1076.317,362.670,-99.575,175.682,30.117,155.329
C02361=1076.324,362.918,-99.612,175.686,30.123,155.330
C02362=1076.330,363.165,-99.648,175.689,30.129,155.331
C02363=1076.337,363.412,-99.685,175.693,30.135,155.332
C02364=1076.343,363.659,-99.722,175.697,30.141,155.334
C02365=1076.349,363.906,-99.759,175.700,30.147,155.335
C02366=1076.356,364.154,-99.796,175.704,30.153,155.336
C02367=1076.362,364.401,-99.832,175.707,30.159,155.337
C02368=1076.369,364.648,-99.869,175.711,30.165,155.338
C02369=1076.375,364.894,-99.906,175.715,30.172,155.339
C02370=1076.381,365.142,-99.943,175.718,30.178,155.341
C02371=1076.388,365.389,-99.980,175.722,30.184,155.342
C02372=1076.393,365.637,-100.017,175.725,30.190,155.343
C02373=1076.400,365.883,-100.054,175.730,30.196,155.344
C02374=1076.406,366.131,-100.091,175.733,30.202,155.345
C02375=1076.413,366.378,-100.128,175.736,30.208,155.346
C02376=1076.418,366.625,-100.165,175.740,30.214,155.348
C02377=1076.425,366.872,-100.202,175.744,30.220,155.349
C02378=1076.432,367.119,-100.239,175.748,30.227,155.350
C02379=1076.438,367.366,-100.276,175.751,30.233,155.351
C02380=1076.444,367.613,-100.313,175.754,30.239,155.352
C02381=1076.451,367.861,-100.351,175.759,30.246,155.354
C02382=1076.457,368.107,-100.388,175.762,30.252,155.355
C02383=1076.463,368.355,-100.425,175.766,30.258,155.356
C02384=1076.470,368.602,-100.463,175.769,30.264,155.357
C02385=1076.476,368.849,-100.500,175.773,30.271,155.359
C02386=1076.482,369.096,-100.537,175.777,30.277,155.360
C02387=1076.489,369.343,-100.575,175.780,30.283,155.361
C02388=1076.495,369.590,-100.611,175.785,30.289,155.362
C02389=1076.501,369.837,-100.649,175.788,30.296,155.363
C02390=1076.508,370.084,-100.687,175.791,30.302,155.365
C02391=1076.514,370.331,-100.724,175.796,30.309,155.366
C02392=1076.521,370.579,-100.761,175.799,30.315,155.367
C02393=1076.527,370.825,-100.799,175.803,30.321,155.368
C02394=1076.533,371.048,-100.832,175.806,30.327,155.369
C02395=1076.538,371.270,-100.867,175.810,30.333,155.371
C02396=1076.545,371.493,-100.900,175.813,30.338,155.372
C02397=1076.551,371.715,-100.934,175.816,30.344,155.373
C02398=1076.556,371.937,-100.968,175.820,30.350,155.374
C02399=1076.562,372.160,-101.001,175.823,30.356,155.375
C02400=1076.568,372.383,-101.036,175.827,30.362,155.376
C02401=1076.574,372.605,-101.069,175.829,30.368,155.377
C02402=1076.580,372.852,-101.107,175.834,30.374,155.379
C02403=1076.587,373.099,-101.145,175.837,30.380,155.380
C02404=1076.594,373.346,-101.183,175.842,30.387,155.381
C02405=1076.600,373.593,-101.220,175.845,30.393,155.382
C02406=1076.607,373.840,-101.258,175.848,30.400,155.384
C02407=1076.613,374.087,-101.296,175.853,30.407,155.385
C02408=1076.619,374.334,-101.334,175.856,30.413,155.386
C02409=1076.625,374.581,-101.372,175.860,30.420,155.388
C02410=1076.632,374.828,-101.410,175.864,30.427,155.389
C02411=1076.639,375.074,-101.448,175.867,30.433,155.390
C02412=1076.645,375.322,-101.486,175.871,30.440,155.392
C02413=1076.651,375.569,-101.523,175.875,30.447,155.393
C02414=1076.657,375.816,-101.562,175.879,30.453,155.394
C02415=1076.663,376.063,-101.599,175.883,30.460,155.396
C02416=1076.670,376.310,-101.638,175.886,30.467,155.397
C02417=1076.677,376.556,-101.675,175.890,30.473,155.398
C02418=1076.683,376.804,-101.713,175.894,30.480,155.400
C02419=1076.690,377.050,-101.752,175.898,30.487,155.401
C02420=1076.696,377.297,-101.790,175.902,30.494,155.402
C02421=1076.703,377.545,-101.828,175.906,30.501,155.404
C02422=1076.709,377.791,-101.867,175.910,30.507,155.405
C02423=1076.715,378.038,-101.905,175.913,30.514,155.406
C02424=1076.722,378.285,-101.944,175.917,30.521,155.408
C02425=1076.729,378.532,-101.982,175.921,30.528,155.409
C02426=1076.736,378.778,-102.020,175.925,30.535,155.410
C02427=1076.742,379.026,-102.058,175.929,30.541,155.412
C02428=1076.749,379.272,-102.097,175.932,30.548,155.413
C02429=1076.755,379.519,-102.134,175.937,30.555,155.415
C02430=1076.762,379.766,-102.173,175.940,30.562,155.416
C02431=1076.768,380.014,-102.211,175.945,30.569,155.417
C02432=1076.775,380.260,-102.250,175.948,30.576,155.419
C02433=1076.781,380.507,-102.288,175.952,30.583,155.420
C02434=1076.788,380.754,-102.327,175.956,30.590,155.421
C02435=1076.794,381.001,-102.366,175.960,30.597,155.423
C02436=1076.801,381.248,-102.404,175.964,30.604,155.424
C02437=1076.807,381.494,-102.442,175.968,30.611,155.426
C02438=1076.814,381.741,-102.481,175.972,30.618,155.427
C02439=1076.821,381.988,-102.520,175.976,30.625,155.428
C02440=1076.827,382.235,-102.558,175.979,30.632,155.430
C02441=1076.834,382.482,-102.597,175.984,30.639,155.431
C02442=1076.840,382.729,-102.636,175.987,30.646,155.433
C02443=1076.846,382.975,-102.675,175.992,30.653,155.434
C02444=1076.853,383.222,-102.713,175.995,30.660,155.436
C02445=1076.860,383.469,-102.752,176.000,30.668,155.437
C02446=1076.867,383.716,-102.791,176.003,30.675,155.439
C02447=1076.872,383.962,-102.830,176.007,30.682,155.440
C02448=1076.879,384.209,-102.869,176.011,30.690,155.442
C02449=1076.886,384.456,-102.908,176.015,30.697,155.443
C02450=1076.892,384.693,-102.946,176.019,30.704,155.444
C02451=1076.898,384.930,-102.983,176.023,30.711,155.446
C02452=1076.905,385.167,-103.020,176.027,30.718,155.447
C02453=1076.910,385.404,-103.058,176.030,30.725,155.449
C02454=1076.918,385.641,-103.095,176.034,30.732,155.450
C02455=1076.923,385.878,-103.133,176.038,30.739,155.451
C02456=1076.930,386.115,-103.170,176.042,30.746,155.453
C02457=1076.936,386.351,-103.208,176.046,30.753,155.454
C02458=1076.943,386.598,-103.247,176.049,30.760,155.456
C02459=1076.950,386.845,-103.286,176.054,30.768,155.457
C02460=1076.956,387.092,-103.325,176.058,30.775,155.459
C02461=1076.963,387.338,-103.365,176.062,30.782,155.460
C02462=1076.970,387.585,-103.404,176.066,30.790,155.462
C02463=1076.976,387.832,-103.443,176.070,30.797,155.463
C02464=1076.983,388.078,-103.483,176.074,30.805,155.465
C02465=1076.990,388.325,-103.521,176.078,30.812,155.466
C02466=1076.996,388.572,-103.561,176.082,30.820,155.468
C02467=1077.003,388.819,-103.600,176.086,30.827,155.470
C02468=1077.010,389.065,-103.639,176.091,30.835,155.471
C02469=1077.016,389.312,-103.679,176.094,30.842,155.473
C02470=1077.023,389.559,-103.718,176.098,30.850,155.474
C02471=1077.029,389.805,-103.758,176.103,30.858,155.476
C02472=1077.037,390.053,-103.798,176.106,30.865,155.477
C02473=1077.044,390.299,-103.837,176.111,30.873,155.479
C02474=1077.050,390.546,-103.877,176.115,30.880,155.480
C02475=1077.057,390.792,-103.916,176.119,30.888,155.482
C02476=1077.063,391.039,-103.956,176.123,30.896,155.484
C02477=1077.070,391.286,-103.995,176.128,30.903,155.485
C02478=1077.077,391.532,-104.035,176.131,30.911,155.487
C02479=1077.084,391.778,-104.075,176.135,30.919,155.488
C02480=1077.090,392.026,-104.115,176.140,30.927,155.490
C02481=1077.097,392.272,-104.154,176.144,30.934,155.492
C02482=1077.104,392.519,-104.194,176.148,30.942,155.493
C02483=1077.110,392.765,-104.235,176.152,30.950,155.495
C02484=1077.117,393.012,-104.274,176.157,30.958,155.496
C02485=1077.124,393.259,-104.314,176.160,30.966,155.498
C02486=1077.130,393.506,-104.354,176.165,30.974,155.500
C02487=1077.137,393.752,-104.394,176.169,30.982,155.501
C02488=1077.144,393.999,-104.434,176.174,30.989,155.503
C02489=1077.150,394.245,-104.474,176.177,30.997,155.505
C02490=1077.158,394.492,-104.514,176.181,31.005,155.506
C02491=1077.164,394.739,-104.554,176.186,31.013,155.508
C02492=1077.171,394.985,-104.594,176.190,31.022,155.510
C02493=1077.178,395.232,-104.635,176.194,31.029,155.511
C02494=1077.185,395.479,-104.674,176.198,31.037,155.513
C02495=1077.191,395.725,-104.714,176.203,31.046,155.515
C02496=1077.197,395.972,-104.754,176.207,31.054,155.516
C02497=1077.205,396.218,-104.796,176.211,31.062,155.518
C02498=1077.211,396.465,-104.836,176.215,31.070,155.520
C02499=1077.218,396.711,-104.876,176.220,31.079,155.522
C02500=1077.225,396.958,-104.916,176.224,31.087,155.523
C02501=1077.232,397.205,-104.956,176.229,31.095,155.525
C02502=1077.239,397.451,-104.997,176.232,31.103,155.527
C02503=1077.245,397.698,-105.037,176.237,31.111,155.528
C02504=1077.252,397.944,-105.078,176.241,31.120,155.530
C02505=1077.259,398.191,-105.119,176.245,31.128,155.532
C02506=1077.266,398.436,-105.159,176.250,31.136,155.534
C02507=1077.272,398.679,-105.199,176.253,31.144,155.535
C02508=1077.279,398.924,-105.239,176.258,31.153,155.537
C02509=1077.286,399.168,-105.279,176.262,31.161,155.539
C02510=1077.293,399.412,-105.319,176.267,31.169,155.541
C02511=1077.300,399.657,-105.360,176.271,31.178,155.542
C02512=1077.307,399.901,-105.400,176.275,31.186,155.544
C02513=1077.312,400.145,-105.440,176.279,31.194,155.546
C02514=1077.320,400.392,-105.482,176.284,31.203,155.548
C02515=1077.326,400.638,-105.522,176.288,31.212,155.550
C02516=1077.333,400.885,-105.563,176.293,31.220,155.551
C02517=1077.340,401.131,-105.604,176.297,31.229,155.553
C02518=1077.347,401.378,-105.644,176.302,31.237,155.555
C02519=1077.354,401.625,-105.686,176.305,31.245,155.557
C02520=1077.361,401.871,-105.726,176.310,31.254,155.559
C02521=1077.368,402.117,-105.768,176.314,31.263,155.561
C02522=1077.375,402.364,-105.808,176.319,31.271,155.562
C02523=1077.381,402.611,-105.850,176.323,31.280,155.564
C02524=1077.388,402.857,-105.891,176.328,31.289,155.566
C02525=1077.395,403.103,-105.932,176.332,31.298,155.568
C02526=1077.402,403.350,-105.973,176.337,31.306,155.570
C02527=1077.410,403.596,-106.014,176.341,31.315,155.572
C02528=1077.416,403.843,-106.054,176.346,31.324,155.574
C02529=1077.423,404.090,-106.096,176.350,31.333,155.576
C02530=1077.430,404.336,-106.137,176.355,31.342,155.577
C02531=1077.437,404.583,-106.179,176.359,31.351,155.579
C02532=1077.444,404.829,-106.219,176.364,31.360,155.581
C02533=1077.450,405.076,-106.261,176.368,31.368,155.583
C02534=1077.458,405.322,-106.303,176.373,31.377,155.585
C02535=1077.465,405.568,-106.344,176.377,31.387,155.587
C02536=1077.471,405.815,-106.386,176.382,31.396,155.589
C02537=1077.479,406.061,-106.427,176.386,31.405,155.591
C02538=1077.485,406.308,-106.469,176.391,31.414,155.593
C02539=1077.492,406.555,-106.510,176.395,31.423,155.595
C02540=1077.499,406.800,-106.552,176.400,31.432,155.597
C02541=1077.506,407.047,-106.594,176.405,31.441,155.599
C02542=1077.513,407.293,-106.635,176.409,31.450,155.601
C02543=1077.520,407.540,-106.677,176.414,31.460,155.603
C02544=1077.527,407.786,-106.719,176.418,31.469,155.605
C02545=1077.534,408.033,-106.760,176.423,31.478,155.607
C02546=1077.541,408.278,-106.802,176.427,31.488,155.609
C02547=1077.547,408.525,-106.844,176.433,31.497,155.611
C02548=1077.554,408.772,-106.886,176.437,31.506,155.613
C02549=1077.562,409.018,-106.928,176.442,31.516,155.615
C02550=1077.568,409.265,-106.970,176.446,31.525,155.617
C02551=1077.576,409.511,-107.011,176.451,31.535,155.619
C02552=1077.583,409.757,-107.054,176.455,31.544,155.621
C02553=1077.590,410.003,-107.096,176.460,31.553,155.623
C02554=1077.597,410.250,-107.138,176.465,31.563,155.625
C02555=1077.604,410.497,-107.180,176.470,31.573,155.627
C02556=1077.611,410.743,-107.222,176.475,31.582,155.629
C02557=1077.618,410.989,-107.264,176.479,31.591,155.631
C02558=1077.625,411.236,-107.307,176.484,31.601,155.634
C02559=1077.632,411.482,-107.348,176.488,31.611,155.636
C02560=1077.639,411.728,-107.391,176.494,31.620,155.638
C02561=1077.647,411.974,-107.433,176.499,31.630,155.640
C02562=1077.653,412.220,-107.475,176.503,31.640,155.642
C02563=1077.660,412.465,-107.517,176.508,31.650,155.644
C02564=1077.667,412.711,-107.559,176.513,31.659,155.646
C02565=1077.675,412.956,-107.602,176.518,31.669,155.648
C02566=1077.682,413.202,-107.643,176.522,31.679,155.650
C02567=1077.688,413.448,-107.686,176.527,31.689,155.653
C02568=1077.696,413.693,-107.728,176.533,31.699,155.655
C02569=1077.703,413.939,-107.770,176.537,31.709,155.657
C02570=1077.710,414.185,-107.813,176.542,31.718,155.659
C02571=1077.717,414.430,-107.856,176.546,31.728,155.661
C02572=1077.724,414.677,-107.899,176.552,31.738,155.663
C02573=1077.732,414.923,-107.941,176.557,31.748,155.666
C02574=1077.739,415.170,-107.983,176.561,31.758,155.668
C02575=1077.746,415.416,-108.026,176.567,31.768,155.670
C02576=1077.753,415.662,-108.069,176.571,31.778,155.672
C02577=1077.761,415.909,-108.112,176.576,31.789,155.675
C02578=1077.768,416.155,-108.155,176.582,31.799,155.677
C02579=1077.775,416.401,-108.198,176.586,31.809,155.679
C02580=1077.782,416.647,-108.240,176.592,31.819,155.681
C02581=1077.789,416.893,-108.284,176.597,31.829,155.684
C02582=1077.796,417.140,-108.327,176.601,31.840,155.686
C02583=1077.803,417.385,-108.370,176.607,31.850,155.688
C02584=1077.810,417.632,-108.412,176.612,31.860,155.691
C02585=1077.818,417.878,-108.456,176.617,31.871,155.693
C02586=1077.825,418.124,-108.499,176.622,31.881,155.695
C02587=1077.832,418.370,-108.542,176.626,31.891,155.697
C02588=1077.840,418.616,-108.585,176.632,31.902,155.700
C02589=1077.847,418.862,-108.628,176.637,31.913,155.702
C02590=1077.854,419.109,-108.672,176.642,31.923,155.705
C02591=1077.862,419.355,-108.715,176.647,31.934,155.707
C02592=1077.868,419.601,-108.757,176.653,31.945,155.709
C02593=1077.876,419.847,-108.801,176.657,31.955,155.712
C02594=1077.883,420.093,-108.844,176.663,31.966,155.714
C02595=1077.891,420.339,-108.888,176.668,31.976,155.716
C02596=1077.898,420.585,-108.931,176.673,31.987,155.719
C02597=1077.906,420.831,-108.975,176.678,31.998,155.721
C02598=1077.912,421.077,-109.019,176.684,32.009,155.724
C02599=1077.920,421.324,-109.062,176.689,32.020,155.726
C02600=1077.927,421.569,-109.106,176.694,32.031,155.729
C02601=1077.935,421.816,-109.149,176.700,32.042,155.731
C02602=1077.942,422.061,-109.192,176.705,32.052,155.733
C02603=1077.949,422.308,-109.237,176.710,32.063,155.736
C02604=1077.957,422.554,-109.280,176.715,32.074,155.738
C02605=1077.964,422.800,-109.324,176.721,32.086,155.741
C02606=1077.971,423.045,-109.368,176.726,32.097,155.743
C02607=1077.979,423.292,-109.412,176.731,32.107,155.746
C02608=1077.987,423.538,-109.455,176.737,32.119,155.748
C02609=1077.993,423.783,-109.500,176.743,32.130,155.751
C02610=1078.001,424.030,-109.543,176.747,32.141,155.754
C02611=1078.007,424.276,-109.587,176.753,32.153,155.756
C02612=1078.016,424.521,-109.632,176.759,32.164,155.759
C02613=1078.023,424.768,-109.675,176.764,32.175,155.761
C02614=1078.030,425.013,-109.720,176.769,32.186,155.764
C02615=1078.038,425.260,-109.763,176.775,32.198,155.766
C02616=1078.045,425.506,-109.808,176.780,32.209,155.769
C02617=1078.053,425.751,-109.853,176.786,32.221,155.772
C02618=1078.061,426.013,-109.899,176.791,32.233,155.774
C02619=1078.069,426.276,-109.947,176.797,32.245,155.777
C02620=1078.077,426.538,-109.994,176.804,32.258,155.780
C02621=1078.085,426.799,-110.041,176.810,32.270,155.783
C02622=1078.092,427.046,-110.085,176.815,32.282,155.785
C02623=1078.100,427.292,-110.130,176.820,32.293,155.788
C02624=1078.108,427.538,-110.174,176.826,32.305,155.791
C02625=1078.115,427.784,-110.219,176.832,32.317,155.793
C02626=1078.123,428.029,-110.263,176.838,32.329,155.796
C02627=1078.130,428.275,-110.308,176.843,32.341,155.799
C02628=1078.138,428.521,-110.353,176.848,32.352,155.802
C02629=1078.145,428.767,-110.397,176.854,32.364,155.804
C02630=1078.153,429.013,-110.442,176.860,32.376,155.807
C02631=1078.161,429.258,-110.487,176.866,32.388,155.810
C02632=1078.168,429.504,-110.532,176.872,32.400,155.813
C02633=1078.175,429.750,-110.577,176.877,32.412,155.815
C02634=1078.182,429.996,-110.621,176.883,32.424,155.818
C02635=1078.190,430.241,-110.666,176.889,32.437,155.821
C02636=1078.198,430.487,-110.711,176.895,32.449,155.824
C02637=1078.205,430.733,-110.756,176.900,32.461,155.827
C02638=1078.213,430.978,-110.801,176.906,32.473,155.829
C02639=1078.221,431.224,-110.846,176.912,32.486,155.832
C02640=1078.228,431.470,-110.891,176.917,32.498,155.835
C02641=1078.236,431.716,-110.937,176.923,32.510,155.838
C02642=1078.244,431.962,-110.981,176.929,32.523,155.841
C02643=1078.252,432.208,-111.027,176.935,32.535,155.844
C02644=1078.259,432.454,-111.072,176.941,32.548,155.847
C02645=1078.267,432.699,-111.118,176.947,32.560,155.849
C02646=1078.275,432.945,-111.163,176.953,32.573,155.852
C02647=1078.282,433.191,-111.208,176.959,32.586,155.855
C02648=1078.290,433.436,-111.254,176.965,32.598,155.858
C02649=1078.297,433.681,-111.299,176.971,32.611,155.861
C02650=1078.305,433.927,-111.345,176.978,32.624,155.864
C02651=1078.313,434.172,-111.391,176.984,32.637,155.867
C02652=1078.321,434.419,-111.436,176.989,32.649,155.870
C02653=1078.328,434.665,-111.482,176.995,32.663,155.873
C02654=1078.336,434.910,-111.527,177.001,32.675,155.876
C02655=1078.343,435.155,-111.573,177.007,32.688,155.879
C02656=1078.351,435.401,-111.619,177.013,32.701,155.882
C02657=1078.359,435.647,-111.665,177.019,32.714,155.885
C02658=1078.367,435.892,-111.710,177.025,32.727,155.889
C02659=1078.375,436.137,-111.757,177.032,32.741,155.892
C02660=1078.383,436.383,-111.802,177.038,32.754,155.895
C02661=1078.391,436.629,-111.848,177.044,32.767,155.898
C02662=1078.398,436.874,-111.894,177.050,32.780,155.901
C02663=1078.406,437.120,-111.940,177.056,32.794,155.904
C02664=1078.414,437.365,-111.987,177.063,32.807,155.907
C02665=1078.422,437.611,-112.033,177.070,32.820,155.910
C02666=1078.430,437.857,-112.079,177.076,32.834,155.913
C02667=1078.438,438.102,-112.125,177.083,32.847,155.917
C02668=1078.445,438.347,-112.171,177.089,32.861,155.920
C02669=1078.454,438.593,-112.217,177.095,32.874,155.923
C02670=1078.462,438.838,-112.263,177.101,32.888,155.926
C02671=1078.470,439.084,-112.310,177.108,32.902,155.930
C02672=1078.478,439.330,-112.357,177.114,32.915,155.933
C02673=1078.486,439.575,-112.403,177.120,32.929,155.936
C02674=1078.497,439.941,-112.472,177.130,32.950,155.941
C02675=1078.510,440.308,-112.542,177.140,32.970,155.946
C02676=1078.521,440.674,-112.612,177.150,32.992,155.951
C02677=1078.533,441.039,-112.681,177.160,33.013,155.956
C02678=1078.542,441.285,-112.728,177.166,33.027,155.959
C02679=1078.549,441.531,-112.775,177.172,33.041,155.963
C02680=1078.557,441.776,-112.822,177.180,33.055,155.966
C02681=1078.565,442.021,-112.869,177.186,33.069,155.969
C02682=1078.574,442.267,-112.916,177.193,33.084,155.973
C02683=1078.581,442.512,-112.963,177.199,33.098,155.976
C02684=1078.589,442.758,-113.009,177.206,33.113,155.980
C02685=1078.597,443.003,-113.057,177.213,33.127,155.983
C02686=1078.606,443.248,-113.104,177.220,33.141,155.987
C02687=1078.613,443.493,-113.151,177.226,33.156,155.990
C02688=1078.622,443.739,-113.198,177.233,33.171,155.994
C02689=1078.630,443.984,-113.246,177.241,33.185,155.997
C02690=1078.639,444.230,-113.293,177.247,33.200,156.001
C02691=1078.646,444.474,-113.340,177.254,33.215,156.004
C02692=1078.655,444.720,-113.387,177.261,33.230,156.008
C02693=1078.663,444.965,-113.435,177.268,33.244,156.011
C02694=1078.670,445.211,-113.482,177.275,33.260,156.015
C02695=1078.679,445.456,-113.530,177.282,33.275,156.019
C02696=1078.687,445.701,-113.578,177.289,33.290,156.022
C02697=1078.696,445.946,-113.626,177.296,33.305,156.026
C02698=1078.704,446.191,-113.673,177.303,33.320,156.030
C02699=1078.712,446.436,-113.720,177.310,33.335,156.033
C02700=1078.720,446.681,-113.768,177.316,33.350,156.037
C02701=1078.728,446.926,-113.816,177.323,33.365,156.041
C02702=1078.737,447.171,-113.864,177.328,33.381,156.045
C02703=1078.745,447.416,-113.912,177.335,33.396,156.048
C02704=1078.754,447.662,-113.960,177.340,33.411,156.052
C02705=1078.762,447.908,-114.008,177.346,33.426,156.056
C02706=1078.771,448.152,-114.056,177.350,33.441,156.059
C02707=1078.779,448.398,-114.104,177.355,33.456,156.063
C02708=1078.787,448.643,-114.152,177.360,33.471,156.067
C02709=1078.795,448.887,-114.201,177.364,33.486,156.071
C02710=1078.805,449.132,-114.248,177.368,33.501,156.074
C02711=1078.815,449.377,-114.295,177.373,33.515,156.078
C02712=1078.827,449.623,-114.341,177.376,33.528,156.081
C02713=1078.841,449.869,-114.386,177.381,33.541,156.085
C02714=1078.478,449.864,-114.613,177.357,33.704,156.128
C02715=1078.459,449.535,-114.553,177.351,33.687,156.123
C02716=1078.444,449.207,-114.491,177.345,33.669,156.119
C02717=1078.431,448.882,-114.427,177.340,33.649,156.114
C02718=1078.420,448.556,-114.363,177.334,33.629,156.109
C02719=1078.412,448.311,-114.315,177.329,33.614,156.105
C02720=1078.403,448.066,-114.268,177.324,33.599,156.102
C02721=1078.395,447.821,-114.220,177.318,33.584,156.098
C02722=1078.387,447.575,-114.172,177.313,33.569,156.094
C02723=1078.379,447.330,-114.124,177.307,33.554,156.090
C02724=1078.371,447.086,-114.075,177.302,33.539,156.087
C02725=1078.362,446.841,-114.027,177.295,33.523,156.083
C02726=1078.354,446.595,-113.979,177.288,33.508,156.079
C02727=1078.346,446.350,-113.932,177.282,33.493,156.075
C02728=1078.337,446.105,-113.885,177.275,33.478,156.072
C02729=1078.329,445.860,-113.836,177.267,33.463,156.068
C02730=1078.321,445.614,-113.788,177.261,33.448,156.064
C02731=1078.313,445.369,-113.740,177.253,33.433,156.061
C02732=1078.304,445.124,-113.693,177.246,33.418,156.057
C02733=1078.296,444.878,-113.646,177.239,33.403,156.053
C02734=1078.288,444.633,-113.598,177.232,33.388,156.050
C02735=1078.279,444.388,-113.550,177.224,33.373,156.046
C02736=1078.271,444.143,-113.503,177.218,33.359,156.043
C02737=1078.263,443.898,-113.456,177.211,33.343,156.039
C02738=1078.255,443.653,-113.408,177.204,33.329,156.036
C02739=1078.246,443.408,-113.361,177.197,33.315,156.032
C02740=1078.239,443.162,-113.314,177.190,33.300,156.029
C02741=1078.230,442.916,-113.267,177.183,33.285,156.025
C02742=1078.222,442.672,-113.219,177.176,33.271,156.022
C02743=1078.214,442.426,-113.173,177.170,33.256,156.018
C02744=1078.206,442.180,-113.125,177.162,33.242,156.015
C02745=1078.198,441.936,-113.079,177.156,33.228,156.011
C02746=1078.190,441.690,-113.032,177.150,33.213,156.008
C02747=1078.181,441.445,-112.984,177.142,33.199,156.004
C02748=1078.173,441.199,-112.937,177.136,33.185,156.001
C02749=1078.166,440.954,-112.890,177.129,33.171,155.998
C02750=1078.157,440.709,-112.844,177.123,33.157,155.994
C02751=1078.149,440.441,-112.793,177.115,33.142,155.991
C02752=1078.140,440.173,-112.742,177.108,33.127,155.987
C02753=1078.131,439.906,-112.691,177.101,33.111,155.983
C02754=1078.123,439.637,-112.640,177.094,33.096,155.980
C02755=1078.115,439.392,-112.594,177.087,33.082,155.977
C02756=1078.107,439.146,-112.548,177.080,33.069,155.973
C02757=1078.099,438.901,-112.501,177.074,33.055,155.970
C02758=1078.091,438.656,-112.454,177.068,33.041,155.967
C02759=1078.083,438.410,-112.408,177.061,33.028,155.964
C02760=1078.075,438.165,-112.362,177.055,33.014,155.960
C02761=1078.066,437.919,-112.316,177.048,33.001,155.957
C02762=1078.058,437.674,-112.269,177.042,32.987,155.954
C02763=1078.051,437.428,-112.223,177.035,32.974,155.951
C02764=1078.042,437.183,-112.177,177.029,32.961,155.948
C02765=1078.035,436.937,-112.131,177.023,32.947,155.944
C02766=1078.027,436.691,-112.085,177.017,32.934,155.941
C02767=1078.019,436.446,-112.038,177.010,32.920,155.938
C02768=1078.011,436.201,-111.992,177.004,32.908,155.935
C02769=1078.003,435.955,-111.946,176.997,32.894,155.932
C02770=1077.996,435.709,-111.901,176.991,32.881,155.929
C02771=1077.988,435.464,-111.855,176.985,32.868,155.926
C02772=1077.980,435.218,-111.809,176.979,32.855,155.923
C02773=1077.972,434.972,-111.764,176.972,32.842,155.920
C02774=1077.964,434.727,-111.718,176.966,32.829,155.917
C02775=1077.957,434.481,-111.672,176.960,32.816,155.914
C02776=1077.949,434.236,-111.627,176.954,32.803,155.911
C02777=1077.941,433.990,-111.581,176.948,32.791,155.908
C02778=1077.933,433.744,-111.535,176.942,32.778,155.905
C02779=1077.926,433.499,-111.489,176.936,32.765,155.902
C02780=1077.918,433.253,-111.444,176.930,32.752,155.899
C02781=1077.910,433.008,-111.398,176.924,32.740,155.896
C02782=1077.903,432.762,-111.353,176.918,32.727,155.893
C02783=1077.895,432.517,-111.307,176.912,32.714,155.890
C02784=1077.888,432.271,-111.262,176.906,32.702,155.887
C02785=1077.880,432.024,-111.216,176.900,32.689,155.884
C02786=1077.871,431.779,-111.171,176.894,32.677,155.881
C02787=1077.864,431.533,-111.126,176.888,32.665,155.878
C02788=1077.857,431.288,-111.081,176.882,32.652,155.876
C02789=1077.849,431.042,-111.036,176.876,32.640,155.873
C02790=1077.841,430.797,-110.991,176.870,32.628,155.870
C02791=1077.833,430.550,-110.946,176.864,32.615,155.867
C02792=1077.826,430.304,-110.901,176.858,32.603,155.864
C02793=1077.819,430.059,-110.855,176.852,32.591,155.861
C02794=1077.810,429.813,-110.811,176.846,32.579,155.859
C02795=1077.803,429.567,-110.766,176.840,32.567,155.856
C02796=1077.796,429.321,-110.721,176.835,32.555,155.853
C02797=1077.787,429.076,-110.676,176.830,32.543,155.850
C02798=1077.780,428.830,-110.631,176.824,32.530,155.847
C02799=1077.773,428.584,-110.586,176.818,32.519,155.845
C02800=1077.765,428.339,-110.542,176.812,32.507,155.842
C02801=1077.758,428.093,-110.497,176.806,32.495,155.839
C02802=1077.751,427.847,-110.452,176.801,32.483,155.837
C02803=1077.743,427.601,-110.408,176.795,32.471,155.834
C02804=1077.735,427.355,-110.363,176.789,32.460,155.831
C02805=1077.727,427.109,-110.319,176.783,32.448,155.829
C02806=1077.720,426.863,-110.274,176.778,32.437,155.826
C02807=1077.711,426.600,-110.227,176.772,32.424,155.823
C02808=1077.704,426.336,-110.179,176.766,32.412,155.820
C02809=1077.696,426.073,-110.132,176.760,32.399,155.817
C02810=1077.688,425.809,-110.084,176.754,32.387,155.815
C02811=1077.680,425.563,-110.040,176.748,32.376,155.812
C02812=1077.673,425.317,-109.996,176.743,32.364,155.809
C02813=1077.665,425.071,-109.951,176.738,32.353,155.807
C02814=1077.657,424.825,-109.908,176.732,32.341,155.804
C02815=1077.650,424.579,-109.863,176.726,32.330,155.802
C02816=1077.642,424.333,-109.820,176.720,32.319,155.799
C02817=1077.636,424.087,-109.775,176.716,32.307,155.796
C02818=1077.628,423.841,-109.731,176.710,32.296,155.794
C02819=1077.620,423.595,-109.687,176.705,32.285,155.791
C02820=1077.613,423.349,-109.643,176.699,32.274,155.789
C02821=1077.606,423.103,-109.600,176.693,32.263,155.786
C02822=1077.598,422.858,-109.556,176.689,32.251,155.784
C02823=1077.591,422.611,-109.511,176.683,32.240,155.781
C02824=1077.583,422.365,-109.468,176.677,32.229,155.779
C02825=1077.576,422.119,-109.424,176.672,32.218,155.776
C02826=1077.569,421.873,-109.380,176.666,32.207,155.774
C02827=1077.562,421.627,-109.336,176.662,32.196,155.771
C02828=1077.554,421.381,-109.293,176.656,32.185,155.769
C02829=1077.547,421.135,-109.249,176.651,32.175,155.766
C02830=1077.540,420.889,-109.205,176.645,32.164,155.764
C02831=1077.533,420.643,-109.162,176.641,32.153,155.762
C02832=1077.525,420.397,-109.118,176.635,32.142,155.759
C02833=1077.518,420.151,-109.075,176.629,32.132,155.757
C02834=1077.510,419.905,-109.031,176.624,32.121,155.754
C02835=1077.503,419.659,-108.988,176.619,32.110,155.752
C02836=1077.495,419.412,-108.945,176.614,32.100,155.750
C02837=1077.488,419.166,-108.902,176.609,32.089,155.747
C02838=1077.480,418.920,-108.858,176.603,32.079,155.745
C02839=1077.473,418.674,-108.815,176.599,32.068,155.743
C02840=1077.466,418.427,-108.772,176.593,32.057,155.740
C02841=1077.459,418.182,-108.729,176.588,32.047,155.738
C02842=1077.451,417.936,-108.686,176.583,32.037,155.736
C02843=1077.444,417.689,-108.643,176.578,32.026,155.733
C02844=1077.437,417.443,-108.600,176.572,32.016,155.731
C02845=1077.430,417.198,-108.556,176.568,32.005,155.729
C02846=1077.422,416.951,-108.513,176.563,31.995,155.726
C02847=1077.415,416.705,-108.470,176.557,31.985,155.724
C02848=1077.408,416.459,-108.428,176.552,31.975,155.722
C02849=1077.401,416.213,-108.384,176.548,31.965,155.720
C02850=1077.394,415.966,-108.341,176.542,31.954,155.717
C02851=1077.387,415.720,-108.299,176.537,31.944,155.715
C02852=1077.380,415.474,-108.256,176.533,31.934,155.713
C02853=1077.373,415.228,-108.213,176.527,31.924,155.711
C02854=1077.365,414.981,-108.170,176.522,31.914,155.708
C02855=1077.358,414.735,-108.127,176.518,31.903,155.706
C02856=1077.350,414.489,-108.085,176.512,31.893,155.704
C02857=1077.344,414.243,-108.042,176.507,31.884,155.702
C02858=1077.336,413.996,-108.000,176.503,31.874,155.699
C02859=1077.329,413.750,-107.957,176.497,31.864,155.697
C02860=1077.322,413.504,-107.915,176.492,31.854,155.695
C02861=1077.315,413.257,-107.873,176.488,31.844,155.693
C02862=1077.308,413.012,-107.829,176.483,31.834,155.691
C02863=1077.300,412.766,-107.787,176.477,31.825,155.689
C02864=1077.293,412.520,-107.745,176.473,31.815,155.687
C02865=1077.285,412.273,-107.703,176.468,31.805,155.684
C02866=1077.279,412.026,-107.661,176.464,31.796,155.682
C02867=1077.272,411.780,-107.618,176.458,31.785,155.680
C02868=1077.264,411.534,-107.576,176.453,31.776,155.678
C02869=1077.257,411.287,-107.534,176.449,31.767,155.676
C02870=1077.250,411.041,-107.491,176.444,31.757,155.674
C02871=1077.243,410.795,-107.449,176.439,31.747,155.672
C02872=1077.236,410.548,-107.407,176.434,31.738,155.670
C02873=1077.229,410.302,-107.365,176.429,31.728,155.668
C02874=1077.222,410.056,-107.323,176.425,31.719,155.665
C02875=1077.215,409.810,-107.280,176.420,31.709,155.663
C02876=1077.208,409.563,-107.239,176.415,31.700,155.661
C02877=1077.201,409.317,-107.197,176.411,31.691,155.659
C02878=1077.194,409.070,-107.155,176.406,31.681,155.657
C02879=1077.187,408.824,-107.113,176.400,31.671,155.655
C02880=1077.180,408.577,-107.071,176.396,31.662,155.653
C02881=1077.173,408.332,-107.029,176.391,31.653,155.651
C02882=1077.167,408.085,-106.988,176.387,31.643,155.649
C02883=1077.159,407.839,-106.946,176.382,31.634,155.647
C02884=1077.152,407.592,-106.904,176.377,31.625,155.645
C02885=1077.145,407.346,-106.862,176.373,31.616,155.643
C02886=1077.138,407.099,-106.820,176.368,31.606,155.641
C02887=1077.131,406.853,-106.779,176.364,31.597,155.639
C02888=1077.125,406.607,-106.737,176.359,31.588,155.637
C02889=1077.117,406.360,-106.695,176.355,31.579,155.635
C02890=1077.111,406.113,-106.654,176.350,31.570,155.633
C02891=1077.104,405.867,-106.612,176.345,31.561,155.631
C02892=1077.096,405.621,-106.570,176.341,31.552,155.629
C02893=1077.090,405.375,-106.529,176.336,31.542,155.627
C02894=1077.083,405.128,-106.488,176.332,31.534,155.625
C02895=1077.075,404.881,-106.446,176.327,31.525,155.623
C02896=1077.069,404.635,-106.405,176.323,31.516,155.621
C02897=1077.062,404.389,-106.364,176.318,31.507,155.620
C02898=1077.055,404.142,-106.323,176.313,31.498,155.618
C02899=1077.048,403.895,-106.281,176.309,31.489,155.616
C02900=1077.041,403.649,-106.240,176.304,31.480,155.614
C02901=1077.034,403.403,-106.199,176.300,31.472,155.612
C02902=1077.027,403.156,-106.157,176.295,31.463,155.610
C02903=1077.020,402.910,-106.116,176.291,31.454,155.608
C02904=1077.013,402.664,-106.075,176.286,31.445,155.606
C02905=1077.007,402.417,-106.034,176.281,31.437,155.605
C02906=1076.999,402.170,-105.992,176.277,31.428,155.603
C02907=1076.993,401.924,-105.952,176.272,31.419,155.601
C02908=1076.986,401.677,-105.911,176.269,31.411,155.599
C02909=1076.978,401.430,-105.870,176.264,31.402,155.597
C02910=1076.972,401.185,-105.829,176.260,31.393,155.595
C02911=1076.965,400.937,-105.788,176.255,31.385,155.593
C02912=1076.958,400.691,-105.747,176.251,31.376,155.592
C02913=1076.951,400.445,-105.706,176.246,31.368,155.590
C02914=1076.945,400.198,-105.665,176.242,31.359,155.588
C02915=1076.937,399.953,-105.624,176.237,31.351,155.586
C02916=1076.930,399.708,-105.585,176.233,31.342,155.584
C02917=1076.924,399.463,-105.544,176.229,31.334,155.583
C02918=1076.917,399.219,-105.503,176.224,31.325,155.581
C02919=1076.911,398.973,-105.463,176.220,31.317,155.579
C02920=1076.904,398.728,-105.423,176.215,31.309,155.577
C02921=1076.897,398.483,-105.383,176.212,31.301,155.576
C02922=1076.891,398.239,-105.342,176.207,31.293,155.574
C02923=1076.883,397.992,-105.302,176.203,31.284,155.572
C02924=1076.876,397.745,-105.262,176.198,31.275,155.570
C02925=1076.869,397.499,-105.220,176.194,31.267,155.569
C02926=1076.863,397.252,-105.180,176.190,31.259,155.567
C02927=1076.856,397.005,-105.140,176.186,31.251,155.565
C02928=1076.849,396.758,-105.099,176.181,31.243,155.563
C02929=1076.843,396.512,-105.059,176.177,31.234,155.562
C02930=1076.836,396.265,-105.018,176.173,31.227,155.560
C02931=1076.829,396.019,-104.979,176.169,31.219,155.558
C02932=1076.822,395.773,-104.938,176.164,31.210,155.557
C02933=1076.815,395.525,-104.898,176.160,31.202,155.555
C02934=1076.809,395.279,-104.857,176.156,31.194,155.553
C02935=1076.802,395.033,-104.817,176.152,31.186,155.551
C02936=1076.794,394.786,-104.777,176.147,31.178,155.550
C02937=1076.788,394.539,-104.737,176.143,31.170,155.548
C02938=1076.782,394.293,-104.697,176.139,31.162,155.546
C02939=1076.775,394.046,-104.657,176.135,31.154,155.545
C02940=1076.768,393.800,-104.617,176.130,31.146,155.543
C02941=1076.761,393.553,-104.576,176.126,31.138,155.541
C02942=1076.755,393.307,-104.536,176.122,31.130,155.540
C02943=1076.748,393.060,-104.497,176.118,31.122,155.538
C02944=1076.741,392.812,-104.457,176.113,31.114,155.537
C02945=1076.735,392.566,-104.417,176.110,31.107,155.535
C02946=1076.728,392.320,-104.377,176.105,31.098,155.533
C02947=1076.721,392.073,-104.337,176.101,31.091,155.532
C02948=1076.714,391.827,-104.298,176.097,31.083,155.530
C02949=1076.707,391.579,-104.258,176.093,31.075,155.528
C02950=1076.701,391.333,-104.218,176.088,31.067,155.527
C02951=1076.694,391.087,-104.178,176.085,31.060,155.525
C02952=1076.688,390.839,-104.139,176.080,31.052,155.524
C02953=1076.681,390.593,-104.099,176.076,31.044,155.522
C02954=1076.674,390.347,-104.060,176.072,31.037,155.520
C02955=1076.667,390.099,-104.020,176.068,31.029,155.519
C02956=1076.660,389.853,-103.980,176.063,31.022,155.517
C02957=1076.654,389.606,-103.941,176.060,31.014,155.516
C02958=1076.647,389.360,-103.901,176.055,31.006,155.514
C02959=1076.639,389.113,-103.862,176.051,30.999,155.513
C02960=1076.633,388.866,-103.822,176.047,30.991,155.511
C02961=1076.627,388.619,-103.783,176.043,30.984,155.510
C02962=1076.619,388.373,-103.744,176.038,30.976,155.508
C02963=1076.613,388.126,-103.704,176.035,30.969,155.506
C02964=1076.606,387.880,-103.665,176.030,30.961,155.505
C02965=1076.599,387.633,-103.626,176.027,30.954,155.503
C02966=1076.593,387.386,-103.587,176.022,30.947,155.502
C02967=1076.586,387.140,-103.547,176.018,30.939,155.500
C02968=1076.579,386.893,-103.508,176.014,30.932,155.499
C02969=1076.573,386.646,-103.469,176.010,30.924,155.497
C02970=1076.566,386.400,-103.429,176.006,30.917,155.496
C02971=1076.560,386.161,-103.392,176.002,30.910,155.494
C02972=1076.554,385.923,-103.354,175.998,30.903,155.493
C02973=1076.547,385.686,-103.316,175.994,30.896,155.492
C02974=1076.541,385.449,-103.279,175.990,30.889,155.490
C02975=1076.535,385.211,-103.241,175.987,30.882,155.489
C02976=1076.528,384.973,-103.204,175.982,30.875,155.487
C02977=1076.522,384.736,-103.166,175.979,30.868,155.486
C02978=1076.516,384.498,-103.128,175.975,30.860,155.484
C02979=1076.509,384.251,-103.089,175.971,30.853,155.483
C02980=1076.503,384.005,-103.051,175.967,30.846,155.481
C02981=1076.496,383.759,-103.012,175.963,30.839,155.480
C02982=1076.490,383.511,-102.972,175.959,30.832,155.479
C02983=1076.483,383.265,-102.934,175.955,30.824,155.477
C02984=1076.476,383.018,-102.895,175.951,30.817,155.476
C02985=1076.469,382.771,-102.856,175.947,30.810,155.474
C02986=1076.464,382.525,-102.817,175.943,30.803,155.473
C02987=1076.457,382.278,-102.778,175.939,30.796,155.471
C02988=1076.450,382.031,-102.739,175.935,30.788,155.470
C02989=1076.444,381.783,-102.701,175.931,30.782,155.468
C02990=1076.437,381.537,-102.663,175.927,30.774,155.467
C02991=1076.431,381.290,-102.624,175.923,30.767,155.466
C02992=1076.424,381.044,-102.585,175.919,30.760,155.464
C02993=1076.417,380.796,-102.547,175.916,30.753,155.463
C02994=1076.410,380.549,-102.508,175.911,30.746,155.461
C02995=1076.404,380.303,-102.469,175.908,30.740,155.460
C02996=1076.398,380.056,-102.431,175.904,30.733,155.459
C02997=1076.391,379.809,-102.393,175.900,30.726,155.457
C02998=1076.384,379.562,-102.354,175.896,30.719,155.456
C02999=1076.378,379.315,-102.316,175.892,30.712,155.454
C03000=1076.371,379.069,-102.277,175.888,30.705,155.453
C03001=1076.365,378.821,-102.239,175.884,30.698,155.452
C03002=1076.357,378.575,-102.201,175.880,30.691,155.450
C03003=1076.351,378.328,-102.163,175.876,30.685,155.449
C03004=1076.345,378.081,-102.124,175.873,30.678,155.447
C03005=1076.338,377.834,-102.086,175.869,30.671,155.446
C03006=1076.332,377.588,-102.048,175.865,30.664,155.445
C03007=1076.325,377.340,-102.009,175.861,30.658,155.443
C03008=1076.319,377.093,-101.971,175.857,30.650,155.442
C03009=1076.313,376.846,-101.933,175.853,30.644,155.441
C03010=1076.306,376.599,-101.895,175.850,30.637,155.439
C03011=1076.300,376.352,-101.857,175.845,30.630,155.438
C03012=1076.293,376.106,-101.819,175.842,30.623,155.437
C03013=1076.286,375.858,-101.781,175.837,30.617,155.435
C03014=1076.280,375.612,-101.743,175.834,30.610,155.434
C03015=1076.274,375.364,-101.705,175.831,30.603,155.433
C03016=1076.268,375.118,-101.666,175.826,30.597,155.431
C03017=1076.261,374.871,-101.628,175.823,30.590,155.430
C03018=1076.254,374.624,-101.591,175.819,30.584,155.429
C03019=1076.248,374.377,-101.553,175.815,30.577,155.427
C03020=1076.241,374.129,-101.515,175.811,30.570,155.426
C03021=1076.236,373.883,-101.477,175.807,30.564,155.425
C03022=1076.229,373.635,-101.439,175.803,30.557,155.424
C03023=1076.222,373.389,-101.402,175.800,30.551,155.422
C03024=1076.216,373.141,-101.364,175.796,30.544,155.421
C03025=1076.210,372.894,-101.326,175.792,30.538,155.420
C03026=1076.203,372.647,-101.288,175.789,30.531,155.418
C03027=1076.197,372.424,-101.254,175.785,30.525,155.417
C03028=1076.191,372.202,-101.220,175.782,30.519,155.416
C03029=1076.185,371.979,-101.186,175.778,30.514,155.415
C03030=1076.179,371.755,-101.152,175.775,30.508,155.414
C03031=1076.174,371.532,-101.118,175.771,30.502,155.413
C03032=1076.168,371.309,-101.084,175.768,30.496,155.412
C03033=1076.162,371.086,-101.051,175.764,30.490,155.410
C03034=1076.156,370.862,-101.016,175.762,30.485,155.409
C03035=1076.150,370.616,-100.979,175.757,30.478,155.408
C03036=1076.143,370.369,-100.941,175.754,30.472,155.407
C03037=1076.137,370.122,-100.904,175.750,30.466,155.406
C03038=1076.131,369.875,-100.867,175.746,30.459,155.404
C03039=1076.124,369.628,-100.829,175.742,30.453,155.403
C03040=1076.118,369.381,-100.791,175.739,30.446,155.402
C03041=1076.111,369.133,-100.755,175.735,30.440,155.401
C03042=1076.105,368.886,-100.717,175.731,30.434,155.399
C03043=1076.098,368.640,-100.680,175.728,30.428,155.398
C03044=1076.092,368.392,-100.642,175.724,30.421,155.397
C03045=1076.085,368.146,-100.605,175.720,30.415,155.396
C03046=1076.079,367.897,-100.568,175.716,30.409,155.395
C03047=1076.073,367.651,-100.531,175.713,30.403,155.393
C03048=1076.067,367.404,-100.494,175.710,30.396,155.392
C03049=1076.060,367.156,-100.456,175.705,30.390,155.391
C03050=1076.053,366.909,-100.420,175.702,30.383,155.390
C03051=1076.047,366.663,-100.382,175.698,30.377,155.388
C03052=1076.041,366.416,-100.345,175.695,30.371,155.387
C03053=1076.035,366.168,-100.307,175.690,30.365,155.386
C03054=1076.028,365.921,-100.271,175.687,30.359,155.385
C03055=1076.023,365.674,-100.234,175.684,30.353,155.384
C03056=1076.016,365.427,-100.197,175.680,30.347,155.383
C03057=1076.009,365.180,-100.160,175.677,30.340,155.381
C03058=1076.003,364.932,-100.123,175.672,30.334,155.380
C03059=1075.997,364.686,-100.086,175.669,30.328,155.379
C03060=1075.991,364.439,-100.049,175.665,30.322,155.378
C03061=1075.984,364.191,-100.012,175.662,30.316,155.377
C03062=1075.978,363.944,-99.975,175.658,30.310,155.375
C03063=1075.971,363.697,-99.938,175.654,30.304,155.374
C03064=1075.965,363.450,-99.902,175.651,30.298,155.373
C03065=1075.958,363.202,-99.865,175.647,30.292,155.372
C03066=1075.952,362.955,-99.828,175.644,30.286,155.371
C03067=1075.946,362.708,-99.791,175.640,30.280,155.370
C03068=1075.940,362.461,-99.755,175.636,30.274,155.369
C03069=1075.933,362.213,-99.718,175.632,30.268,155.367
C03070=1075.927,361.966,-99.682,175.629,30.262,155.366
C03071=1075.920,361.719,-99.645,175.626,30.256,155.365
C03072=1075.914,361.472,-99.609,175.622,30.250,155.364
C03073=1075.908,361.225,-99.572,175.618,30.244,155.363
C03074=1075.902,360.978,-99.535,175.614,30.239,155.362
C03075=1075.895,360.730,-99.499,175.611,30.233,155.361
C03076=1075.889,360.483,-99.462,175.607,30.227,155.359
C03077=1075.882,360.236,-99.426,175.604,30.221,155.358
C03078=1075.876,359.989,-99.389,175.601,30.215,155.357
C03079=1075.870,359.742,-99.353,175.597,30.209,155.356
C03080=1075.863,359.495,-99.316,175.593,30.203,155.355
C03081=1075.857,359.247,-99.280,175.589,30.197,155.354
C03082=1075.851,359.000,-99.244,175.586,30.191,155.353
C03083=1075.845,358.785,-99.212,175.583,30.187,155.352
C03084=1075.840,358.570,-99.181,175.580,30.182,155.351
C03085=1075.834,358.355,-99.149,175.576,30.177,155.350
C03086=1075.829,358.141,-99.118,175.574,30.171,155.349
C03087=1075.823,357.926,-99.086,175.570,30.166,155.348
C03088=1075.817,357.711,-99.055,175.568,30.161,155.347
C03089=1075.812,357.495,-99.023,175.564,30.157,155.346
C03090=1075.807,357.282,-98.992,175.561,30.152,155.345
C03091=1075.800,357.033,-98.956,175.557,30.145,155.344
C03092=1075.794,356.786,-98.919,175.554,30.140,155.343
C03093=1075.787,356.539,-98.883,175.550,30.134,155.342
C03094=1075.781,356.291,-98.847,175.547,30.128,155.341
C03095=1075.775,356.044,-98.811,175.544,30.123,155.340
C03096=1075.769,355.797,-98.775,175.540,30.117,155.339
C03097=1075.763,355.550,-98.738,175.537,30.111,155.338
C03098=1075.757,355.302,-98.703,175.533,30.106,155.337
C03099=1075.750,355.055,-98.666,175.530,30.100,155.336
C03100=1075.744,354.808,-98.631,175.526,30.095,155.335
C03101=1075.738,354.561,-98.595,175.522,30.089,155.333
C03102=1075.732,354.314,-98.559,175.519,30.083,155.332
C03103=1075.725,354.066,-98.523,175.515,30.078,155.331
C03104=1075.719,353.819,-98.487,175.512,30.072,155.330
C03105=1075.713,353.571,-98.451,175.508,30.067,155.329
C03106=1075.707,353.324,-98.415,175.505,30.060,155.328
C03107=1075.700,353.077,-98.380,175.502,30.055,155.327
C03108=1075.694,352.829,-98.344,175.498,30.049,155.326
C03109=1075.688,352.582,-98.308,175.495,30.044,155.325
C03110=1075.682,352.334,-98.272,175.491,30.038,155.324
C03111=1075.675,352.087,-98.237,175.488,30.033,155.323
C03112=1075.669,351.839,-98.201,175.484,30.027,155.322
C03113=1075.663,351.593,-98.165,175.481,30.022,155.321
C03114=1075.657,351.346,-98.130,175.478,30.016,155.320
C03115=1075.651,351.098,-98.094,175.474,30.011,155.319
C03116=1075.645,350.850,-98.058,175.471,30.006,155.318
C03117=1075.638,350.603,-98.023,175.467,30.000,155.317
C03118=1075.632,350.355,-97.987,175.464,29.995,155.316
C03119=1075.625,350.108,-97.952,175.460,29.989,155.315
C03120=1075.619,349.861,-97.916,175.457,29.984,155.314
C03121=1075.613,349.614,-97.881,175.454,29.979,155.313
C03122=1075.606,349.366,-97.845,175.450,29.973,155.312
C03123=1075.600,349.119,-97.810,175.447,29.967,155.311
C03124=1075.594,348.871,-97.774,175.443,29.962,155.310
C03125=1075.588,348.624,-97.739,175.440,29.956,155.309
C03126=1075.582,348.377,-97.703,175.436,29.951,155.308
C03127=1075.575,348.129,-97.668,175.433,29.946,155.307
C03128=1075.570,347.881,-97.633,175.430,29.940,155.306
C03129=1075.563,347.634,-97.598,175.426,29.935,155.305
C03130=1075.557,347.387,-97.563,175.423,29.930,155.304
C03131=1075.551,347.139,-97.528,175.419,29.924,155.303
C03132=1075.545,346.892,-97.492,175.416,29.919,155.302
C03133=1075.538,346.644,-97.457,175.412,29.914,155.301
C03134=1075.532,346.397,-97.421,175.409,29.908,155.300
C03135=1075.526,346.149,-97.387,175.406,29.903,155.299
C03136=1075.520,345.902,-97.351,175.402,29.897,155.298
C03137=1075.513,345.654,-97.316,175.399,29.892,155.297
C03138=1075.508,345.407,-97.281,175.395,29.887,155.296
C03139=1075.502,345.194,-97.251,175.393,29.882,155.295
C03140=1075.497,344.981,-97.220,175.389,29.878,155.295
C03141=1075.492,344.767,-97.190,175.387,29.873,155.294
C03142=1075.486,344.555,-97.160,175.384,29.869,155.293
C03143=1075.482,344.341,-97.130,175.381,29.864,155.292
C03144=1075.476,344.128,-97.099,175.378,29.860,155.291
C03145=1075.470,343.915,-97.070,175.375,29.855,155.290
C03146=1075.465,343.702,-97.040,175.372,29.851,155.290
C03147=1075.459,343.454,-97.004,175.369,29.846,155.289
C03148=1075.453,343.207,-96.970,175.365,29.840,155.288
C03149=1075.446,342.959,-96.935,175.362,29.835,155.287
C03150=1075.440,342.711,-96.901,175.359,29.830,155.286
C03151=1075.434,342.464,-96.865,175.355,29.825,155.285
C03152=1075.428,342.216,-96.831,175.352,29.819,155.284
C03153=1075.421,341.969,-96.796,175.349,29.815,155.283
C03154=1075.415,341.722,-96.762,175.346,29.809,155.282
C03155=1075.409,341.474,-96.726,175.342,29.804,155.281
C03156=1075.403,341.227,-96.692,175.339,29.799,155.280
C03157=1075.397,340.979,-96.657,175.336,29.794,155.279
C03158=1075.390,340.731,-96.623,175.332,29.789,155.278
C03159=1075.385,340.484,-96.588,175.329,29.784,155.277
C03160=1075.378,340.236,-96.553,175.325,29.779,155.277
C03161=1075.372,339.989,-96.519,175.322,29.773,155.275
C03162=1075.366,339.741,-96.484,175.319,29.768,155.275
C03163=1075.360,339.494,-96.449,175.316,29.763,155.274
C03164=1075.354,339.246,-96.414,175.313,29.758,155.273
C03165=1075.348,338.999,-96.380,175.309,29.753,155.272
C03166=1075.342,338.751,-96.346,175.306,29.748,155.271
C03167=1075.336,338.504,-96.311,175.302,29.743,155.270
C03168=1075.329,338.256,-96.277,175.299,29.737,155.269
C03169=1075.324,338.009,-96.242,175.296,29.732,155.268
C03170=1075.317,337.761,-96.208,175.293,29.727,155.267
C03171=1075.312,337.513,-96.174,175.290,29.722,155.266
C03172=1075.305,337.265,-96.139,175.286,29.717,155.265
C03173=1075.299,337.019,-96.104,175.283,29.713,155.265
C03174=1075.293,336.771,-96.070,175.279,29.708,155.264
C03175=1075.287,336.523,-96.036,175.276,29.703,155.263
C03176=1075.280,336.275,-96.002,175.273,29.698,155.262
C03177=1075.274,336.028,-95.968,175.270,29.693,155.261
C03178=1075.268,335.780,-95.933,175.267,29.688,155.260
C03179=1075.262,335.533,-95.899,175.263,29.683,155.259
C03180=1075.256,335.285,-95.865,175.260,29.677,155.258
C03181=1075.250,335.038,-95.831,175.256,29.673,155.258
C03182=1075.243,334.791,-95.797,175.254,29.668,155.257
C03183=1075.237,334.543,-95.763,175.251,29.663,155.256
C03184=1075.231,334.295,-95.729,175.247,29.658,155.255
C03185=1075.225,334.047,-95.695,175.244,29.653,155.254
C03186=1075.219,333.800,-95.661,175.240,29.648,155.253
C03187=1075.213,333.552,-95.627,175.238,29.643,155.252
C03188=1075.206,333.304,-95.592,175.234,29.638,155.251
C03189=1075.201,333.057,-95.558,175.231,29.633,155.250
C03190=1075.194,332.809,-95.524,175.228,29.628,155.250
C03191=1075.189,332.561,-95.491,175.224,29.624,155.249
C03192=1075.183,332.314,-95.457,175.222,29.619,155.248
C03193=1075.176,332.066,-95.422,175.218,29.614,155.247
C03194=1075.170,331.819,-95.388,175.215,29.609,155.246
C03195=1075.165,331.603,-95.360,175.212,29.605,155.245
C03196=1075.160,331.387,-95.330,175.209,29.600,155.245
C03197=1075.154,331.171,-95.300,175.206,29.596,155.244
C03198=1075.149,330.956,-95.271,175.204,29.592,155.243
C03199=1075.143,330.739,-95.242,175.201,29.588,155.242
C03200=1075.138,330.525,-95.212,175.198,29.584,155.242
C03201=1075.132,330.308,-95.183,175.195,29.579,155.241
C03202=1075.127,330.092,-95.153,175.193,29.576,155.240
C03203=1075.121,329.845,-95.120,175.189,29.571,155.239
C03204=1075.115,329.597,-95.086,175.186,29.566,155.239
C03205=1075.108,329.349,-95.052,175.183,29.561,155.238
C03206=1075.102,329.101,-95.019,175.180,29.556,155.237
C03207=1075.096,328.854,-94.986,175.177,29.552,155.236
C03208=1075.089,328.606,-94.952,175.173,29.547,155.235
C03209=1075.084,328.359,-94.918,175.170,29.542,155.234
C03210=1075.077,328.111,-94.885,175.167,29.538,155.234
C03211=1075.071,327.863,-94.851,175.164,29.533,155.233
C03212=1075.065,327.615,-94.818,175.161,29.528,155.232
C03213=1075.059,327.368,-94.785,175.157,29.524,155.231
C03214=1075.052,327.121,-94.751,175.155,29.519,155.230
C03215=1075.046,326.872,-94.718,175.151,29.514,155.230
C03216=1075.040,326.625,-94.684,175.148,29.510,155.229
C03217=1075.034,326.377,-94.651,175.145,29.505,155.228
C03218=1075.028,326.129,-94.618,175.142,29.500,155.227
C03219=1075.022,325.881,-94.584,175.138,29.495,155.226
C03220=1075.015,325.634,-94.551,175.135,29.490,155.225
C03221=1075.010,325.386,-94.517,175.133,29.486,155.225
C03222=1075.003,325.138,-94.485,175.129,29.481,155.224
C03223=1074.997,324.891,-94.451,175.126,29.476,155.223
C03224=1074.991,324.644,-94.418,175.123,29.472,155.222
C03225=1074.985,324.395,-94.384,175.120,29.467,155.221
C03226=1074.979,324.147,-94.351,175.116,29.463,155.221
C03227=1074.973,323.899,-94.318,175.114,29.458,155.220
C03228=1074.966,323.652,-94.285,175.111,29.453,155.219
C03229=1074.961,323.405,-94.251,175.107,29.449,155.218
C03230=1074.955,323.157,-94.219,175.104,29.444,155.217
C03231=1074.949,322.909,-94.185,175.101,29.439,155.216
C03232=1074.943,322.661,-94.153,175.098,29.435,155.216
C03233=1074.937,322.414,-94.119,175.095,29.430,155.215
C03234=1074.930,322.165,-94.086,175.092,29.426,155.214
C03235=1074.924,321.918,-94.053,175.089,29.421,155.213
C03236=1074.918,321.670,-94.020,175.085,29.416,155.212
C03237=1074.912,321.422,-93.987,175.083,29.412,155.212
C03238=1074.907,321.174,-93.954,175.079,29.407,155.211
C03239=1074.900,320.927,-93.921,175.076,29.402,155.210
C03240=1074.895,320.679,-93.888,175.074,29.398,155.209
C03241=1074.888,320.431,-93.855,175.070,29.393,155.208
C03242=1074.882,320.184,-93.822,175.068,29.389,155.208
C03243=1074.877,319.936,-93.789,175.064,29.384,155.207
C03244=1074.870,319.688,-93.756,175.061,29.379,155.206
C03245=1074.864,319.440,-93.724,175.058,29.375,155.205
C03246=1074.859,319.193,-93.690,175.055,29.370,155.205
C03247=1074.852,318.945,-93.657,175.052,29.365,155.204
C03248=1074.847,318.697,-93.624,175.049,29.361,155.203
C03249=1074.841,318.449,-93.592,175.046,29.356,155.202
C03250=1074.835,318.202,-93.560,175.043,29.352,155.201
C03251=1074.830,317.983,-93.530,175.040,29.348,155.201
C03252=1074.824,317.764,-93.501,175.037,29.344,155.200
C03253=1074.819,317.545,-93.472,175.035,29.340,155.199
C03254=1074.814,317.326,-93.443,175.032,29.336,155.199
C03255=1074.809,317.107,-93.414,175.030,29.332,155.198
C03256=1074.803,316.888,-93.386,175.026,29.327,155.197
C03257=1074.798,316.668,-93.357,175.024,29.323,155.196
C03258=1074.793,316.450,-93.328,175.021,29.320,155.196
C03259=1074.788,316.202,-93.295,175.018,29.315,155.195
C03260=1074.781,315.954,-93.262,175.016,29.311,155.194
C03261=1074.775,315.706,-93.230,175.012,29.306,155.193
C03262=1074.770,315.459,-93.198,175.010,29.302,155.193
C03263=1074.764,315.211,-93.164,175.006,29.297,155.192
C03264=1074.758,314.963,-93.132,175.003,29.292,155.191
C03265=1074.752,314.716,-93.100,175.001,29.287,155.190
C03266=1074.747,314.467,-93.067,174.997,29.283,155.189
C03267=1074.740,314.220,-93.035,174.995,29.279,155.189
C03268=1074.734,313.971,-93.003,174.991,29.274,155.188
C03269=1074.727,313.724,-92.970,174.988,29.270,155.187
C03270=1074.722,313.476,-92.938,174.985,29.266,155.187
C03271=1074.716,313.229,-92.906,174.982,29.261,155.186
C03272=1074.710,312.981,-92.874,174.980,29.257,155.185
C03273=1074.703,312.733,-92.841,174.976,29.253,155.184
C03274=1074.697,312.485,-92.809,174.974,29.248,155.184
C03275=1074.690,312.237,-92.777,174.970,29.244,155.183
C03276=1074.684,311.989,-92.745,174.967,29.239,155.182
C03277=1074.678,311.741,-92.713,174.964,29.235,155.181
C03278=1074.673,311.494,-92.680,174.961,29.231,155.181
C03279=1074.667,311.246,-92.648,174.959,29.226,155.180
C03280=1074.661,310.998,-92.616,174.955,29.222,155.179
C03281=1074.654,310.750,-92.584,174.953,29.218,155.178
C03282=1074.648,310.502,-92.552,174.949,29.213,155.178
C03283=1074.642,310.255,-92.520,174.946,29.209,155.177
C03284=1074.636,310.007,-92.488,174.943,29.204,155.176
C03285=1074.630,309.759,-92.456,174.940,29.200,155.176
C03286=1074.623,309.511,-92.424,174.937,29.196,155.175
C03287=1074.617,309.263,-92.392,174.934,29.191,155.174
C03288=1074.612,309.015,-92.361,174.932,29.187,155.173
C03289=1074.606,308.768,-92.328,174.928,29.183,155.173
C03290=1074.600,308.519,-92.296,174.926,29.178,155.172
C03291=1074.593,308.272,-92.265,174.922,29.174,155.171
C03292=1074.587,308.024,-92.233,174.919,29.170,155.170
C03293=1074.581,307.776,-92.201,174.917,29.165,155.170
C03294=1074.576,307.528,-92.169,174.913,29.161,155.169
C03295=1074.569,307.280,-92.138,174.911,29.157,155.168
C03296=1074.563,307.033,-92.105,174.907,29.153,155.168
C03297=1074.557,306.785,-92.073,174.905,29.148,155.167
C03298=1074.552,306.537,-92.041,174.901,29.144,155.166
C03299=1074.545,306.289,-92.010,174.899,29.140,155.165
C03300=1074.539,306.041,-91.978,174.896,29.135,155.165
C03301=1074.534,305.794,-91.946,174.893,29.131,155.164
C03302=1074.527,305.546,-91.915,174.890,29.127,155.163
C03303=1074.522,305.298,-91.883,174.887,29.122,155.162
C03304=1074.516,305.050,-91.851,174.884,29.118,155.162
C03305=1074.510,304.802,-91.819,174.881,29.114,155.161
C03306=1074.503,304.554,-91.788,174.878,29.109,155.160
C03307=1074.499,304.337,-91.760,174.876,29.106,155.160
C03308=1074.493,304.120,-91.732,174.873,29.102,155.159
C03309=1074.488,303.902,-91.705,174.871,29.098,155.158
C03310=1074.483,303.685,-91.677,174.868,29.094,155.158
C03311=1074.478,303.467,-91.649,174.866,29.091,155.157
C03312=1074.472,303.250,-91.621,174.863,29.087,155.157
C03313=1074.467,303.033,-91.594,174.861,29.083,155.156
C03314=1074.462,302.815,-91.566,174.858,29.079,155.155
C03315=1074.456,302.568,-91.535,174.855,29.075,155.155
C03316=1074.450,302.320,-91.503,174.852,29.071,155.154
C03317=1074.445,302.072,-91.472,174.849,29.066,155.153
C03318=1074.439,301.824,-91.440,174.846,29.062,155.152
C03319=1074.433,301.576,-91.409,174.843,29.058,155.152
C03320=1074.426,301.328,-91.377,174.841,29.053,155.151
C03321=1074.421,301.080,-91.346,174.837,29.049,155.150
C03322=1074.415,300.832,-91.314,174.835,29.045,155.150
C03323=1074.409,300.585,-91.283,174.831,29.041,155.149
C03324=1074.404,300.336,-91.252,174.829,29.036,155.148
C03325=1074.397,300.089,-91.221,174.826,29.032,155.147
C03326=1074.391,299.840,-91.189,174.823,29.028,155.147
C03327=1074.386,299.592,-91.158,174.821,29.024,155.146
C03328=1074.380,299.345,-91.127,174.817,29.019,155.145
C03329=1074.374,299.097,-91.095,174.815,29.015,155.145
C03330=1074.368,298.849,-91.064,174.811,29.010,155.144
C03331=1074.362,298.601,-91.032,174.809,29.007,155.143
C03332=1074.357,298.353,-91.001,174.806,29.002,155.142
C03333=1074.351,298.106,-90.970,174.803,28.997,155.142
C03334=1074.346,297.857,-90.939,174.801,28.994,155.141
C03335=1074.339,297.609,-90.908,174.797,28.989,155.140
C03336=1074.334,297.361,-90.877,174.795,28.985,155.140
C03337=1074.328,297.113,-90.846,174.792,28.981,155.139
C03338=1074.323,296.865,-90.815,174.789,28.976,155.138
C03339=1074.316,296.617,-90.783,174.786,28.972,155.138
C03340=1074.310,296.370,-90.753,174.783,28.968,155.137
C03341=1074.304,296.121,-90.722,174.781,28.964,155.136
C03342=1074.298,295.874,-90.690,174.777,28.960,155.135
C03343=1074.292,295.625,-90.660,174.775,28.956,155.135
C03344=1074.286,295.377,-90.629,174.772,28.952,155.134
C03345=1074.281,295.130,-90.598,174.769,28.947,155.133
C03346=1074.274,294.881,-90.567,174.766,28.943,155.133
C03347=1074.268,294.633,-90.537,174.763,28.939,155.132
C03348=1074.262,294.385,-90.505,174.761,28.935,155.131
C03349=1074.257,294.137,-90.474,174.758,28.931,155.131
C03350=1074.251,293.889,-90.444,174.755,28.927,155.130
C03351=1074.244,293.641,-90.413,174.752,28.923,155.129
C03352=1074.238,293.394,-90.382,174.749,28.918,155.129
C03353=1074.233,293.146,-90.351,174.747,28.914,155.128
C03354=1074.227,292.897,-90.321,174.743,28.910,155.127
C03355=1074.221,292.645,-90.289,174.741,28.906,155.127
C03356=1074.214,292.393,-90.258,174.738,28.902,155.126
C03357=1074.208,292.140,-90.227,174.735,28.898,155.125
C03358=1074.203,291.888,-90.196,174.733,28.894,155.125
C03359=1074.196,291.640,-90.165,174.729,28.889,155.124
C03360=1074.190,291.392,-90.134,174.727,28.885,155.123
C03361=1074.185,291.144,-90.104,174.724,28.881,155.123
C03362=1074.179,290.896,-90.073,174.721,28.877,155.122
C03363=1074.169,290.481,-90.022,174.716,28.870,155.121
C03364=1074.159,290.064,-89.971,174.712,28.863,155.120
C03365=1074.150,289.649,-89.920,174.707,28.856,155.118
C03366=1074.139,289.233,-89.869,174.702,28.849,155.117
C03367=1074.133,288.985,-89.838,174.700,28.845,155.117
C03368=1074.128,288.737,-89.808,174.697,28.841,155.116
C03369=1074.121,288.489,-89.777,174.694,28.837,155.115
C03370=1074.115,288.241,-89.747,174.691,28.833,155.115
C03371=1074.109,287.993,-89.717,174.689,28.829,155.114
C03372=1074.103,287.744,-89.687,174.685,28.825,155.113
C03373=1074.098,287.496,-89.656,174.683,28.821,155.113
C03374=1074.092,287.248,-89.626,174.681,28.817,155.112
C03375=1074.086,287.001,-89.596,174.677,28.813,155.111
C03376=1074.079,286.753,-89.566,174.675,28.809,155.111
C03377=1074.073,286.505,-89.535,174.672,28.805,155.110
C03378=1074.067,286.256,-89.505,174.669,28.801,155.109
C03379=1074.062,286.008,-89.475,174.667,28.797,155.109
C03380=1074.056,285.760,-89.445,174.664,28.793,155.108
C03381=1074.050,285.513,-89.414,174.661,28.788,155.107
C03382=1074.044,285.264,-89.384,174.658,28.785,155.107
C03383=1074.038,285.016,-89.354,174.656,28.781,155.106
C03384=1074.032,284.768,-89.324,174.653,28.776,155.105
C03385=1074.026,284.520,-89.293,174.650,28.772,155.105
C03386=1074.020,284.272,-89.264,174.648,28.768,155.104
C03387=1074.014,284.024,-89.234,174.644,28.764,155.103
C03388=1074.008,283.775,-89.204,174.642,28.760,155.103
C03389=1074.002,283.527,-89.174,174.639,28.756,155.102
C03390=1073.997,283.279,-89.143,174.636,28.752,155.102
C03391=1073.991,283.031,-89.114,174.634,28.748,155.101
C03392=1073.985,282.783,-89.083,174.631,28.744,155.100
C03393=1073.979,282.535,-89.054,174.629,28.740,155.100
C03394=1073.973,282.287,-89.024,174.625,28.736,155.099
C03395=1073.967,282.039,-88.993,174.623,28.732,155.098
C03396=1073.962,281.791,-88.964,174.621,28.727,155.097
C03397=1073.956,281.543,-88.933,174.617,28.723,155.097
C03398=1073.951,281.295,-88.904,174.615,28.719,155.096
C03399=1073.944,281.047,-88.874,174.612,28.715,155.096
C03400=1073.938,280.798,-88.844,174.610,28.711,155.095
C03401=1073.932,280.550,-88.814,174.607,28.707,155.094
C03402=1073.927,280.302,-88.784,174.604,28.703,155.094
C03403=1073.920,280.054,-88.755,174.602,28.699,155.093
C03404=1073.915,279.806,-88.725,174.598,28.695,155.092
C03405=1073.909,279.557,-88.695,174.596,28.691,155.092
C03406=1073.903,279.309,-88.666,174.593,28.687,155.091
C03407=1073.897,279.061,-88.636,174.591,28.683,155.090
C03408=1073.891,278.813,-88.607,174.588,28.679,155.090
C03409=1073.885,278.565,-88.576,174.585,28.675,155.089
C03410=1073.879,278.317,-88.547,174.583,28.671,155.088
C03411=1073.873,278.069,-88.518,174.580,28.667,155.088
C03412=1073.868,277.820,-88.488,174.577,28.663,155.087
C03413=1073.862,277.573,-88.458,174.575,28.659,155.087
C03414=1073.856,277.324,-88.429,174.572,28.655,155.086
C03415=1073.845,276.914,-88.380,174.567,28.649,155.085
C03416=1073.837,276.504,-88.331,174.563,28.642,155.084
C03417=1073.826,276.094,-88.282,174.559,28.636,155.083
C03418=1073.817,275.684,-88.234,174.554,28.629,155.082
C03419=1073.811,275.436,-88.204,174.552,28.625,155.081
C03420=1073.805,275.188,-88.175,174.549,28.621,155.080
C03421=1073.799,274.940,-88.145,174.547,28.617,155.080
C03422=1073.793,274.692,-88.116,174.544,28.613,155.079
C03423=1073.787,274.443,-88.086,174.541,28.609,155.078
C03424=1073.781,274.195,-88.057,174.539,28.605,155.078
C03425=1073.776,273.947,-88.028,174.536,28.601,155.077
C03426=1073.769,273.699,-87.999,174.533,28.597,155.077
C03427=1073.764,273.450,-87.969,174.530,28.593,155.076
C03428=1073.758,273.202,-87.940,174.528,28.589,155.075
C03429=1073.752,272.954,-87.910,174.526,28.586,155.075
C03430=1073.746,272.705,-87.881,174.522,28.581,155.074
C03431=1073.740,272.458,-87.853,174.520,28.577,155.073
C03432=1073.735,272.210,-87.823,174.517,28.573,155.073
C03433=1073.728,271.961,-87.794,174.515,28.569,155.072
C03434=1073.722,271.713,-87.765,174.513,28.566,155.071
C03435=1073.717,271.465,-87.735,174.509,28.561,155.071
C03436=1073.710,271.217,-87.706,174.507,28.558,155.070
C03437=1073.705,270.968,-87.676,174.504,28.554,155.070
C03438=1073.699,270.719,-87.648,174.502,28.550,155.069
C03439=1073.693,270.471,-87.619,174.500,28.546,155.068
C03440=1073.688,270.224,-87.590,174.496,28.542,155.068
C03441=1073.682,269.975,-87.561,174.494,28.538,155.067
C03442=1073.675,269.727,-87.532,174.491,28.534,155.066
C03443=1073.669,269.479,-87.503,174.489,28.530,155.066
C03444=1073.664,269.230,-87.474,174.487,28.526,155.065
C03445=1073.658,268.982,-87.445,174.483,28.522,155.065
C03446=1073.652,268.735,-87.416,174.481,28.518,155.064
C03447=1073.646,268.486,-87.387,174.478,28.514,155.063
C03448=1073.641,268.237,-87.358,174.476,28.510,155.063
C03449=1073.634,267.989,-87.329,174.474,28.506,155.062
C03450=1073.628,267.741,-87.300,174.470,28.502,155.061
C03451=1073.622,267.492,-87.272,174.468,28.499,155.061
C03452=1073.616,267.245,-87.243,174.465,28.495,155.060
C03453=1073.611,266.997,-87.213,174.463,28.491,155.060
C03454=1073.605,266.748,-87.185,174.461,28.487,155.059
C03455=1073.599,266.500,-87.156,174.458,28.483,155.058
C03456=1073.592,266.251,-87.127,174.455,28.479,155.058
C03457=1073.587,266.003,-87.099,174.452,28.475,155.057
C03458=1073.582,265.755,-87.069,174.450,28.471,155.056
C03459=1073.576,265.506,-87.041,174.448,28.467,155.056
C03460=1073.569,265.258,-87.012,174.445,28.463,155.055
C03461=1073.564,265.010,-86.984,174.443,28.459,155.055
C03462=1073.558,264.762,-86.955,174.440,28.455,155.054
C03463=1073.552,264.513,-86.927,174.437,28.451,155.053
C03464=1073.546,264.266,-86.898,174.435,28.448,155.053
C03465=1073.541,264.017,-86.869,174.432,28.444,155.052
C03466=1073.535,263.769,-86.840,174.430,28.440,155.051
C03467=1073.525,263.362,-86.794,174.426,28.434,155.050
C03468=1073.515,262.955,-86.748,174.422,28.427,155.049
C03469=1073.505,262.549,-86.701,174.417,28.421,155.048
C03470=1073.495,262.142,-86.654,174.413,28.415,155.047
C03471=1073.489,261.893,-86.625,174.410,28.411,155.047
C03472=1073.484,261.645,-86.597,174.408,28.407,155.046
C03473=1073.477,261.397,-86.568,174.406,28.403,155.046
C03474=1073.471,261.149,-86.541,174.403,28.399,155.045
C03475=1073.465,260.900,-86.512,174.400,28.395,155.044
C03476=1073.459,260.652,-86.484,174.397,28.392,155.044
C03477=1073.453,260.404,-86.455,174.395,28.388,155.043
C03478=1073.447,260.155,-86.427,174.393,28.384,155.043
C03479=1073.442,259.907,-86.399,174.390,28.380,155.042
C03480=1073.435,259.658,-86.371,174.388,28.376,155.041
C03481=1073.429,259.410,-86.342,174.385,28.372,155.041
C03482=1073.423,259.162,-86.314,174.383,28.368,155.040
C03483=1073.418,258.913,-86.286,174.380,28.364,155.040
C03484=1073.412,258.665,-86.258,174.377,28.360,155.039
C03485=1073.406,258.417,-86.230,174.375,28.356,155.038
C03486=1073.399,258.169,-86.201,174.373,28.352,155.038
C03487=1073.393,257.920,-86.173,174.370,28.349,155.037
C03488=1073.388,257.672,-86.145,174.368,28.345,155.037
C03489=1073.382,257.423,-86.117,174.365,28.341,155.036
C03490=1073.375,257.175,-86.089,174.363,28.338,155.035
C03491=1073.370,256.927,-86.061,174.360,28.334,155.035
C03492=1073.364,256.678,-86.033,174.358,28.330,155.034
C03493=1073.359,256.430,-86.005,174.355,28.325,155.033
C03494=1073.352,256.182,-85.977,174.352,28.322,155.033
C03495=1073.346,255.933,-85.949,174.350,28.318,155.032
C03496=1073.341,255.685,-85.921,174.348,28.314,155.032
C03497=1073.335,255.436,-85.892,174.345,28.310,155.031
C03498=1073.329,255.188,-85.865,174.343,28.307,155.030
C03499=1073.323,254.940,-85.837,174.340,28.303,155.030
C03500=1073.318,254.691,-85.809,174.338,28.299,155.029
C03501=1073.312,254.443,-85.780,174.336,28.295,155.028
C03502=1073.306,254.195,-85.753,174.333,28.291,155.028
C03503=1073.300,253.946,-85.725,174.331,28.287,155.027
C03504=1073.294,253.698,-85.697,174.328,28.283,155.027
C03505=1073.288,253.449,-85.668,174.325,28.279,155.026
C03506=1073.282,253.201,-85.641,174.323,28.275,155.025
C03507=1073.276,252.953,-85.613,174.320,28.271,155.025
C03508=1073.271,252.704,-85.585,174.318,28.267,155.024
C03509=1073.265,252.456,-85.558,174.316,28.263,155.024
C03510=1073.259,252.208,-85.530,174.313,28.259,155.023
C03511=1073.253,251.959,-85.501,174.311,28.255,155.022
C03512=1073.248,251.711,-85.473,174.308,28.252,155.022
C03513=1073.241,251.463,-85.446,174.306,28.248,155.021
C03514=1073.236,251.214,-85.418,174.304,28.244,155.020
C03515=1073.230,250.965,-85.390,174.301,28.240,155.020
C03516=1073.224,250.717,-85.363,174.299,28.236,155.019
C03517=1073.218,250.469,-85.334,174.297,28.232,155.019
C03518=1073.213,250.220,-85.307,174.294,28.228,155.018
C03519=1073.203,249.811,-85.262,174.290,28.222,155.017
C03520=1073.194,249.402,-85.216,174.286,28.215,155.016
C03521=1073.185,248.992,-85.171,174.282,28.209,155.015
C03522=1073.175,248.583,-85.125,174.278,28.202,155.014
C03523=1073.170,248.335,-85.097,174.276,28.198,155.013
C03524=1073.164,248.086,-85.070,174.274,28.195,155.013
C03525=1073.158,247.838,-85.042,174.271,28.191,155.012
C03526=1073.153,247.590,-85.014,174.269,28.187,155.011
C03527=1073.147,247.341,-84.987,174.267,28.183,155.011
C03528=1073.141,247.093,-84.959,174.264,28.179,155.010
C03529=1073.135,246.844,-84.932,174.262,28.175,155.009
C03530=1073.130,246.596,-84.904,174.259,28.171,155.009
C03531=1073.123,246.347,-84.877,174.257,28.167,155.008
C03532=1073.118,246.099,-84.849,174.254,28.163,155.008
C03533=1073.112,245.850,-84.822,174.251,28.159,155.007
C03534=1073.105,245.602,-84.795,174.249,28.156,155.007
C03535=1073.100,245.354,-84.768,174.247,28.151,155.006
C03536=1073.094,245.105,-84.740,174.244,28.147,155.005
C03537=1073.089,244.856,-84.713,174.242,28.143,155.005
C03538=1073.083,244.608,-84.686,174.240,28.140,155.004
C03539=1073.077,244.359,-84.658,174.237,28.136,155.003
C03540=1073.071,244.111,-84.631,174.235,28.132,155.003
C03541=1073.065,243.863,-84.604,174.233,28.128,155.002
C03542=1073.060,243.615,-84.577,174.230,28.124,155.002
C03543=1073.054,243.366,-84.550,174.228,28.120,155.001
C03544=1073.048,243.118,-84.522,174.225,28.116,155.000
C03545=1073.043,242.869,-84.495,174.223,28.112,155.000
C03546=1073.036,242.620,-84.468,174.221,28.108,154.999
C03547=1073.030,242.372,-84.441,174.218,28.105,154.999
C03548=1073.025,242.124,-84.413,174.216,28.101,154.998
C03549=1073.019,241.875,-84.386,174.214,28.097,154.997
C03550=1073.013,241.626,-84.360,174.211,28.093,154.997
C03551=1073.007,241.378,-84.332,174.210,28.090,154.996
C03552=1073.001,241.130,-84.306,174.207,28.086,154.995
C03553=1072.996,240.881,-84.278,174.205,28.082,154.995
C03554=1072.990,240.632,-84.251,174.203,28.078,154.994
C03555=1072.984,240.384,-84.225,174.200,28.074,154.994
C03556=1072.977,240.136,-84.197,174.198,28.070,154.993
C03557=1072.972,239.887,-84.170,174.196,28.067,154.992
C03558=1072.966,239.639,-84.143,174.193,28.063,154.992
C03559=1072.961,239.390,-84.117,174.191,28.059,154.991
C03560=1072.954,239.141,-84.090,174.189,28.055,154.991
C03561=1072.949,238.893,-84.063,174.186,28.051,154.990
C03562=1072.943,238.644,-84.036,174.184,28.047,154.989
C03563=1072.937,238.397,-84.009,174.182,28.043,154.989
C03564=1072.930,238.148,-83.982,174.179,28.039,154.988
C03565=1072.925,237.899,-83.955,174.177,28.035,154.988
C03566=1072.919,237.651,-83.929,174.174,28.031,154.987
C03567=1072.914,237.402,-83.901,174.172,28.027,154.986
C03568=1072.908,237.154,-83.875,174.170,28.024,154.986
C03569=1072.902,236.905,-83.848,174.167,28.020,154.985
C03570=1072.896,236.656,-83.821,174.165,28.016,154.984
C03571=1072.886,236.241,-83.777,174.161,28.010,154.984
C03572=1072.876,235.825,-83.732,174.157,28.003,154.982
C03573=1072.867,235.409,-83.687,174.153,27.996,154.981
C03574=1072.858,234.993,-83.642,174.149,27.990,154.980
C03575=1072.851,234.744,-83.615,174.148,27.986,154.980
C03576=1072.845,234.496,-83.589,174.146,27.982,154.979
C03577=1072.840,234.248,-83.562,174.143,27.978,154.978
C03578=1072.834,233.999,-83.536,174.141,27.975,154.978
C03579=1072.828,233.750,-83.510,174.139,27.971,154.977
C03580=1072.823,233.502,-83.483,174.136,27.967,154.977
C03581=1072.817,233.254,-83.456,174.134,27.963,154.976
C03582=1072.811,233.005,-83.430,174.132,27.959,154.976
C03583=1072.805,232.756,-83.403,174.129,27.955,154.975
C03584=1072.799,232.507,-83.377,174.127,27.951,154.974
C03585=1072.793,232.259,-83.350,174.125,27.947,154.974
C03586=1072.787,232.011,-83.324,174.122,27.944,154.973
C03587=1072.781,231.762,-83.297,174.120,27.939,154.972
C03588=1072.776,231.513,-83.271,174.119,27.936,154.972
C03589=1072.770,231.265,-83.245,174.116,27.932,154.971
C03590=1072.764,231.017,-83.218,174.114,27.928,154.971
C03591=1072.759,230.768,-83.192,174.111,27.924,154.970
C03592=1072.753,230.519,-83.166,174.109,27.920,154.969
C03593=1072.747,230.271,-83.139,174.107,27.916,154.969
C03594=1072.742,230.022,-83.113,174.104,27.913,154.968
C03595=1072.735,229.774,-83.087,174.102,27.908,154.968
C03596=1072.729,229.526,-83.060,174.100,27.904,154.967
C03597=1072.723,229.276,-83.034,174.098,27.900,154.966
C03598=1072.718,229.028,-83.007,174.096,27.897,154.966
C03599=1072.711,228.779,-82.982,174.094,27.893,154.965
C03600=1072.706,228.531,-82.955,174.091,27.889,154.964
C03601=1072.700,228.282,-82.929,174.089,27.886,154.964
C03602=1072.694,228.034,-82.903,174.087,27.882,154.963
C03603=1072.688,227.785,-82.877,174.084,27.877,154.963
C03604=1072.682,227.536,-82.851,174.082,27.874,154.962
C03605=1072.677,227.288,-82.824,174.080,27.870,154.961
C03606=1072.670,227.039,-82.799,174.077,27.866,154.961
C03607=1072.665,226.791,-82.772,174.076,27.862,154.960
C03608=1072.659,226.542,-82.746,174.074,27.859,154.960
C03609=1072.653,226.294,-82.720,174.071,27.855,154.959
C03610=1072.647,226.045,-82.694,174.069,27.850,154.958
C03611=1072.642,225.796,-82.668,174.067,27.846,154.958
C03612=1072.635,225.548,-82.642,174.064,27.843,154.957
C03613=1072.630,225.299,-82.616,174.062,27.839,154.957
C03614=1072.624,225.050,-82.590,174.060,27.835,154.956
C03615=1072.618,224.802,-82.564,174.058,27.831,154.955
C03616=1072.612,224.553,-82.538,174.056,27.827,154.955
C03617=1072.606,224.304,-82.512,174.054,27.823,154.954
C03618=1072.600,224.056,-82.486,174.051,27.819,154.954
